LIN {X 0,Y 325.201,Z 458.699,A -85,B 0,C 180,E1 -14842.55,E2 -14842.55} C_VEL
LIN {X 0,Y 325.198,Z 460.508,A -85,B 0,C 180,E1 -14843.797,E2 -14843.797} C_VEL
LIN {X 0,Y 325.238,Z 461.898,A -85,B 0,C 180,E1 -14845.041,E2 -14845.041} C_VEL
LIN {X 0,Y 325.475,Z 463.331,A -85,B 0,C 180,E1 -14847.525,E2 -14847.525} C_VEL
LIN {X 0,Y 325.603,Z 463.425,A -85,B 0,C 180,E1 -14848.763,E2 -14848.763} C_VEL
LIN {X 0,Y 325.577,Z 463.02,A -85,B 0,C 180,E1 -14850,E2 -14850} C_VEL
LIN {X 0,Y 325.621,Z 461.713,A -85,B 0,C 180,E1 -14852.474,E2 -14852.474} C_VEL
LIN {X 0,Y 325.409,Z 460.927,A -85,B 0,C 180,E1 -14853.715,E2 -14853.715} C_VEL
LIN {X 0,Y 325.339,Z 458.485,A -85,B 0,C 180,E1 -14855.579,E2 -14855.579} C_VEL
LIN {X 0,Y 325.419,Z 455.521,A -85,B 0,C 180,E1 -14856.994,E2 -14856.994} C_VEL
LIN {X 0,Y 325.54,Z 450.546,A -85,B 0,C 180,E1 -14858.692,E2 -14858.692} C_VEL
LIN {X 0,Y 325.777,Z 444.462,A -85,B 0,C 180,E1 -14860.252,E2 -14860.252} C_VEL
LIN {X 0,Y 326.095,Z 438.305,A -85,B 0,C 180,E1 -14861.499,E2 -14861.499} C_VEL
LIN {X 0,Y 326.625,Z 429.473,A -85,B 0,C 180,E1 -14862.899,E2 -14862.899} C_VEL
LIN {X 0,Y 326.943,Z 420.656,A -85,B 0,C 180,E1 -14863.995,E2 -14863.995} C_VEL
LIN {X 0,Y 327.306,Z 414.872,A -85,B 0,C 180,E1 -14864.614,E2 -14864.614} C_VEL
LIN {X 0,Y 327.995,Z 404.103,A -85,B 0,C 180,E1 -14865.823,E2 -14865.823} C_VEL
LIN {X 0,Y 328.456,Z 394.191,A -85,B 0,C 180,E1 -14866.71,E2 -14866.71} C_VEL
LIN {X 0,Y 327.545,Z 382.063,A -85,B 0,C 180,E1 -14867.562,E2 -14867.562} C_VEL
LIN {X 0,Y 327.132,Z 375.822,A -85,B 0,C 180,E1 -14867.908,E2 -14867.908} C_VEL
LIN {X 0,Y 327.626,Z 366.768,A -85,B 0,C 180,E1 -14869.042,E2 -14869.042} C_VEL
LIN {X 0,Y 327.17,Z 358.001,A -85,B 0,C 180,E1 -14870.43,E2 -14870.43} C_VEL
LIN {X 0,Y 328.784,Z 345.205,A -85,B 0,C 180,E1 -14874.635,E2 -14874.635} C_VEL
LIN {X 0,Y 330.645,Z 333.295,A -85,B 0,C 180,E1 -14878.571,E2 -14878.571} C_VEL
LIN {X 0,Y 331.363,Z 329.074,A -85,B 0,C 180,E1 -14879.977,E2 -14879.977} C_VEL
LIN {X 0,Y 331.435,Z 327.269,A -85,B 0,C 180,E1 -14880.592,E2 -14880.592} C_VEL
LIN {X 0,Y 329.253,Z 316.724,A -85,B 0,C 180,E1 -14884.447,E2 -14884.447} C_VEL
LIN {X 0,Y 326.968,Z 305.312,A -85,B 0,C 180,E1 -14888.825,E2 -14888.825} C_VEL
LIN {X 0,Y 326.92,Z 305.233,A -85,B 0,C 180,E1 -14891.792,E2 -14891.792} C_VEL
LIN {X 0,Y 327.446,Z 306.47,A -85,B 0,C 180,E1 -14895.096,E2 -14895.096} C_VEL
LIN {X 0,Y 328.262,Z 309.046,A -85,B 0,C 180,E1 -14898.534,E2 -14898.534} C_VEL
LIN {X 0,Y 329.377,Z 312.876,A -85,B 0,C 180,E1 -14902.137,E2 -14902.137} C_VEL
LIN {X 0,Y 330.222,Z 316.406,A -85,B 0,C 180,E1 -14904.925,E2 -14904.925} C_VEL
LIN {X 0,Y 330.999,Z 321.163,A -85,B 0,C 180,E1 -14908.137,E2 -14908.137} C_VEL
LIN {X 0,Y 331.171,Z 324.386,A -85,B 0,C 180,E1 -14910.085,E2 -14910.085} C_VEL
LIN {X 0,Y 330.472,Z 330.636,A -85,B 0,C 180,E1 -14913.473,E2 -14913.473} C_VEL
LIN {X 0,Y 329.774,Z 338.112,A -85,B 0,C 180,E1 -14917.441,E2 -14917.441} C_VEL
LIN {X 0,Y 329.205,Z 345.556,A -85,B 0,C 180,E1 -14921.322,E2 -14921.322} C_VEL
LIN {X 0,Y 328.9,Z 351.017,A -85,B 0,C 180,E1 -14924.127,E2 -14924.127} C_VEL
LIN {X 0,Y 332.084,Z 361.27,A -85,B 0,C 180,E1 -14925.287,E2 -14925.287} C_VEL
LIN {X 0,Y 333.261,Z 367.816,A -85,B 0,C 180,E1 -14926.104,E2 -14926.104} C_VEL
LIN {X 0,Y 332.238,Z 376.783,A -85,B 0,C 180,E1 -14927.226,E2 -14927.226} C_VEL
LIN {X 0,Y 331.076,Z 383.941,A -85,B 0,C 180,E1 -14928.364,E2 -14928.364} C_VEL
LIN {X 0,Y 330.119,Z 389.732,A -85,B 0,C 180,E1 -14929.573,E2 -14929.573} C_VEL
LIN {X 0,Y 329.305,Z 394.315,A -85,B 0,C 180,E1 -14930.788,E2 -14930.788} C_VEL
LIN {X 0,Y 328.522,Z 397.947,A -85,B 0,C 180,E1 -14932.005,E2 -14932.005} C_VEL
LIN {X 0,Y 327.856,Z 400.687,A -85,B 0,C 180,E1 -14933.228,E2 -14933.228} C_VEL
LIN {X 0,Y 326.757,Z 403.34,A -85,B 0,C 180,E1 -14935.063,E2 -14935.063} C_VEL
LIN {X 0,Y 326.193,Z 404.249,A -85,B 0,C 180,E1 -14936.292,E2 -14936.292} C_VEL
LIN {X 0,Y 325.862,Z 404.462,A -85,B 0,C 180,E1 -14937.526,E2 -14937.526} C_VEL
LIN {X 0,Y 325.68,Z 403.978,A -85,B 0,C 180,E1 -14938.762,E2 -14938.762} C_VEL
LIN {X 0,Y 325.531,Z 402.803,A -85,B 0,C 180,E1 -14939.998,E2 -14939.998} C_VEL
LIN {X 0,Y 325.509,Z 399.647,A -85,B 0,C 180,E1 -14941.854,E2 -14941.854} C_VEL
LIN {X 0,Y 325.609,Z 396.615,A -85,B 0,C 180,E1 -14943.092,E2 -14943.092} C_VEL
LIN {X 0,Y 325.781,Z 391.513,A -85,B 0,C 180,E1 -14944.639,E2 -14944.639} C_VEL
LIN {X 0,Y 326.058,Z 386.269,A -85,B 0,C 180,E1 -14945.875,E2 -14945.875} C_VEL
LIN {X 0,Y 326.233,Z 378.87,A -85,B 0,C 180,E1 -14947.237,E2 -14947.237} C_VEL
LIN {X 0,Y 326.433,Z 371.108,A -85,B 0,C 180,E1 -14948.354,E2 -14948.354} C_VEL
LIN {X 0,Y 326.671,Z 362.647,A -85,B 0,C 180,E1 -14949.284,E2 -14949.284} C_VEL
LIN {X 0,Y 326.921,Z 353.507,A -85,B 0,C 180,E1 -14950.058,E2 -14950.058} C_VEL
LIN {X 0,Y 326.042,Z 345.613,A -85,B 0,C 180,E1 -14950.556,E2 -14950.556} C_VEL
LIN {X 0,Y 326.165,Z 337.653,A -85,B 0,C 180,E1 -14954.155,E2 -14954.155} C_VEL
LIN {X 0,Y 326.232,Z 328.045,A -85,B 0,C 180,E1 -14958.578,E2 -14958.578} C_VEL
LIN {X 0,Y 326.347,Z 320.299,A -85,B 0,C 180,E1 -14962.176,E2 -14962.176} C_VEL
LIN {X 0,Y 326.533,Z 313.209,A -85,B 0,C 180,E1 -14965.495,E2 -14965.495} C_VEL
LIN {X 0,Y 326.706,Z 305.841,A -85,B 0,C 180,E1 -14968.946,E2 -14968.946} C_VEL
LIN {X 0,Y 326.794,Z 303.776,A -85,B 0,C 180,E1 -14969.961,E2 -14969.961} C_VEL
LIN {X 0,Y 326.602,Z 303.799,A -85,B 0,C 180,E1 -14974.018,E2 -14974.018} C_VEL
LIN {X 0,Y 326.617,Z 303.802,A -85,B 0,C 180,E1 -14977.236,E2 -14977.236} C_VEL
LIN {X 0,Y 326.538,Z 303.812,A -85,B 0,C 180,E1 -14981.123,E2 -14981.123} C_VEL
LIN {X 0,Y 326.554,Z 303.807,A -85,B 0,C 180,E1 -14983.524,E2 -14983.524} C_VEL
LIN {X 0,Y 326.568,Z 303.808,A -85,B 0,C 180,E1 -14987.027,E2 -14987.027} C_VEL
LIN {X 0,Y 326.604,Z 303.804,A -85,B 0,C 180,E1 -14990.771,E2 -14990.771} C_VEL
LIN {X 0,Y 326.605,Z 303.802,A -85,B 0,C 180,E1 -14994.479,E2 -14994.479} C_VEL
LIN {X 0,Y 326.599,Z 303.8,A -85,B 0,C 180,E1 -14997.454,E2 -14997.454} C_VEL
LIN {X 0,Y 326.651,Z 303.796,A -85,B 0,C 180,E1 -15000.34,E2 -15000.34} C_VEL
LIN {X 0,Y 326.68,Z 303.795,A -85,B 0,C 180,E1 -15004.515,E2 -15004.515} C_VEL
LIN {X 0,Y 326.636,Z 303.8,A -85,B 0,C 180,E1 -15008.544,E2 -15008.544} C_VEL
LIN {X 0,Y 326.733,Z 303.783,A -85,B 0,C 180,E1 -15011.177,E2 -15011.177} C_VEL
LIN {X 0,Y 326.752,Z 303.78,A -85,B 0,C 180,E1 -15015.433,E2 -15015.433} C_VEL
LIN {X 0,Y 326.746,Z 303.782,A -85,B 0,C 180,E1 -15018.838,E2 -15018.838} C_VEL
LIN {X 0,Y 326.902,Z 303.764,A -85,B 0,C 180,E1 -15022.589,E2 -15022.589} C_VEL
LIN {X 0,Y 326.74,Z 303.782,A -85,B 0,C 180,E1 -15025.064,E2 -15025.064} C_VEL
LIN {X 0,Y 326.998,Z 303.751,A -85,B 0,C 180,E1 -15027.536,E2 -15027.536} C_VEL
LIN {X 0,Y 327.016,Z 303.748,A -85,B 0,C 180,E1 -15031.231,E2 -15031.231} C_VEL
LIN {X 0,Y 326.745,Z 303.785,A -85,B 0,C 180,E1 -15033.7,E2 -15033.7} C_VEL
LIN {X 0,Y 326.932,Z 303.761,A -85,B 0,C 180,E1 -15036.17,E2 -15036.17} C_VEL
LIN {X 0,Y 326.771,Z 303.782,A -85,B 0,C 180,E1 -15039.908,E2 -15039.908} C_VEL
LIN {X 0,Y 326.747,Z 303.787,A -85,B 0,C 180,E1 -15043.686,E2 -15043.686} C_VEL
LIN {X 0,Y 326.689,Z 303.793,A -85,B 0,C 180,E1 -15047.529,E2 -15047.529} C_VEL
LIN {X 0,Y 326.657,Z 303.793,A -85,B 0,C 180,E1 -15050.135,E2 -15050.135} C_VEL
LIN {X 0,Y 326.642,Z 303.795,A -85,B 0,C 180,E1 -15054.13,E2 -15054.13} C_VEL
LIN {X 0,Y 326.675,Z 303.791,A -85,B 0,C 180,E1 -15056.859,E2 -15056.859} C_VEL
LIN {X 0,Y 326.629,Z 303.796,A -85,B 0,C 180,E1 -15060.612,E2 -15060.612} C_VEL
LIN {X 0,Y 326.598,Z 303.8,A -85,B 0,C 180,E1 -15064.021,E2 -15064.021} C_VEL
LIN {X 0,Y 326.621,Z 303.802,A -85,B 0,C 180,E1 -15067.24,E2 -15067.24} C_VEL
LIN {X 0,Y 326.57,Z 303.808,A -85,B 0,C 180,E1 -15071.133,E2 -15071.133} C_VEL
LIN {X 0,Y 326.52,Z 303.813,A -85,B 0,C 180,E1 -15074.744,E2 -15074.744} C_VEL
LIN {X 0,Y 326.555,Z 303.805,A -85,B 0,C 180,E1 -15078.154,E2 -15078.154} C_VEL
LIN {X 0,Y 326.575,Z 303.804,A -85,B 0,C 180,E1 -15081.387,E2 -15081.387} C_VEL
LIN {X 0,Y 326.614,Z 303.803,A -85,B 0,C 180,E1 -15084.853,E2 -15084.853} C_VEL
LIN {X 0,Y 326.811,Z 303.868,A -85,B 0,C 180,E1 -15088.48,E2 -15088.48} C_VEL
LIN {X 0,Y 326.946,Z 306.82,A -85,B 0,C 180,E1 -15090.372,E2 -15090.372} C_VEL
LIN {X 0,Y 326.556,Z 312.39,A -85,B 0,C 180,E1 -15093.822,E2 -15093.822} C_VEL
LIN {X 0,Y 326.169,Z 319.095,A -85,B 0,C 180,E1 -15097.9,E2 -15097.9} C_VEL
LIN {X 0,Y 325.915,Z 324.514,A -85,B 0,C 180,E1 -15101.13,E2 -15101.13} C_VEL
LIN {X 0,Y 325.724,Z 328.884,A -85,B 0,C 180,E1 -15103.692,E2 -15103.692} C_VEL
LIN {X 0,Y 325.001,Z 330.075,A -85,B 0,C 180,E1 -15104.347,E2 -15104.347} C_VEL
LIN {X 0,Y 322.085,Z 332.054,A -85,B 0,C 180,E1 -15105.362,E2 -15105.362} C_VEL
LIN {X 0,Y 319.171,Z 334.053,A -85,B 0,C 180,E1 -15106.394,E2 -15106.394} C_VEL
LIN {X 0,Y 318.479,Z 335.258,A -85,B 0,C 180,E1 -15107.067,E2 -15107.067} C_VEL
LIN {X 0,Y 318.465,Z 336.636,A -85,B 0,C 180,E1 -15107.86,E2 -15107.86} C_VEL
LIN {X 0,Y 319.617,Z 348.07,A -85,B 0,C 180,E1 -15108.668,E2 -15108.668} C_VEL
LIN {X 0,Y 320.397,Z 354.645,A -85,B 0,C 180,E1 -15109.256,E2 -15109.256} C_VEL
LIN {X 0,Y 319.903,Z 364.882,A -85,B 0,C 180,E1 -15110.358,E2 -15110.358} C_VEL
LIN {X 0,Y 319.519,Z 374.615,A -85,B 0,C 180,E1 -15111.706,E2 -15111.706} C_VEL
LIN {X 0,Y 319.21,Z 382.258,A -85,B 0,C 180,E1 -15113.047,E2 -15113.047} C_VEL
LIN {X 0,Y 318.893,Z 389.43,A -85,B 0,C 180,E1 -15114.627,E2 -15114.627} C_VEL
LIN {X 0,Y 318.581,Z 395.045,A -85,B 0,C 180,E1 -15116.207,E2 -15116.207} C_VEL
LIN {X 0,Y 318.433,Z 400.056,A -85,B 0,C 180,E1 -15118.104,E2 -15118.104} C_VEL
LIN {X 0,Y 318.484,Z 403.441,A -85,B 0,C 180,E1 -15120.002,E2 -15120.002} C_VEL
LIN {X 0,Y 318.636,Z 404.864,A -85,B 0,C 180,E1 -15121.265,E2 -15121.265} C_VEL
LIN {X 0,Y 318.85,Z 405.644,A -85,B 0,C 180,E1 -15122.528,E2 -15122.528} C_VEL
LIN {X 0,Y 319.196,Z 405.78,A -85,B 0,C 180,E1 -15123.789,E2 -15123.789} C_VEL
LIN {X 0,Y 319.771,Z 405.275,A -85,B 0,C 180,E1 -15125.045,E2 -15125.045} C_VEL
LIN {X 0,Y 320.449,Z 404.147,A -85,B 0,C 180,E1 -15126.297,E2 -15126.297} C_VEL
LIN {X 0,Y 321.74,Z 401.238,A -85,B 0,C 180,E1 -15128.164,E2 -15128.164} C_VEL
LIN {X 0,Y 323.183,Z 396.853,A -85,B 0,C 180,E1 -15130.02,E2 -15130.02} C_VEL
LIN {X 0,Y 324.589,Z 391.903,A -85,B 0,C 180,E1 -15131.555,E2 -15131.555} C_VEL
LIN {X 0,Y 326.271,Z 385.501,A -85,B 0,C 180,E1 -15133.073,E2 -15133.073} C_VEL
LIN {X 0,Y 328.143,Z 377.5,A -85,B 0,C 180,E1 -15134.577,E2 -15134.577} C_VEL
LIN {X 0,Y 329.055,Z 372.691,A -85,B 0,C 180,E1 -15135.338,E2 -15135.338} C_VEL
LIN {X 0,Y 328.549,Z 366.669,A -85,B 0,C 180,E1 -15136.371,E2 -15136.371} C_VEL
LIN {X 0,Y 326.537,Z 357.316,A -85,B 0,C 180,E1 -15137.935,E2 -15137.935} C_VEL
LIN {X 0,Y 323.137,Z 347.004,A -85,B 0,C 180,E1 -15139.608,E2 -15139.608} C_VEL
LIN {X 0,Y 321.875,Z 343.462,A -85,B 0,C 180,E1 -15140.22,E2 -15140.22} C_VEL
LIN {X 0,Y 322.799,Z 339.37,A -85,B 0,C 180,E1 -15143.875,E2 -15143.875} C_VEL
LIN {X 0,Y 323.719,Z 336.122,A -85,B 0,C 180,E1 -15147.125,E2 -15147.125} C_VEL
LIN {X 0,Y 324.569,Z 333.676,A -85,B 0,C 180,E1 -15149.987,E2 -15149.987} C_VEL
LIN {X 0,Y 325.098,Z 331.86,A -85,B 0,C 180,E1 -15152.716,E2 -15152.716} C_VEL
LIN {X 0,Y 325.329,Z 330.489,A -85,B 0,C 180,E1 -15155.683,E2 -15155.683} C_VEL
LIN {X 0,Y 325.489,Z 329.814,A -85,B 0,C 180,E1 -15158.984,E2 -15158.984} C_VEL
LIN {X 0,Y 325.709,Z 329.954,A -85,B 0,C 180,E1 -15161.984,E2 -15161.984} C_VEL
LIN {X 0,Y 326.092,Z 331.016,A -85,B 0,C 180,E1 -15165.336,E2 -15165.336} C_VEL
LIN {X 0,Y 326.701,Z 333.227,A -85,B 0,C 180,E1 -15168.846,E2 -15168.846} C_VEL
LIN {X 0,Y 327.276,Z 335.665,A -85,B 0,C 180,E1 -15171.482,E2 -15171.482} C_VEL
LIN {X 0,Y 328.152,Z 339.585,A -85,B 0,C 180,E1 -15174.672,E2 -15174.672} C_VEL
LIN {X 0,Y 328.855,Z 343.249,A -85,B 0,C 180,E1 -15177.115,E2 -15177.115} C_VEL
LIN {X 0,Y 328.826,Z 345.636,A -85,B 0,C 180,E1 -15178.412,E2 -15178.412} C_VEL
LIN {X 0,Y 326.738,Z 351.583,A -85,B 0,C 180,E1 -15181.055,E2 -15181.055} C_VEL
LIN {X 0,Y 324.056,Z 361.03,A -85,B 0,C 180,E1 -15184.831,E2 -15184.831} C_VEL
LIN {X 0,Y 326.737,Z 372.97,A -85,B 0,C 180,E1 -15185.96,E2 -15185.96} C_VEL
LIN {X 0,Y 328.385,Z 385.404,A -85,B 0,C 180,E1 -15187.189,E2 -15187.189} C_VEL
LIN {X 0,Y 328.621,Z 394.021,A -85,B 0,C 180,E1 -15188.084,E2 -15188.084} C_VEL
LIN {X 0,Y 327.755,Z 404.734,A -85,B 0,C 180,E1 -15189.28,E2 -15189.28} C_VEL
LIN {X 0,Y 325.502,Z 416.387,A -85,B 0,C 180,E1 -15190.776,E2 -15190.776} C_VEL
LIN {X 0,Y 323.559,Z 425.786,A -85,B 0,C 180,E1 -15192.296,E2 -15192.296} C_VEL
LIN {X 0,Y 321.827,Z 434.424,A -85,B 0,C 180,E1 -15194.013,E2 -15194.013} C_VEL
LIN {X 0,Y 320.493,Z 441.391,A -85,B 0,C 180,E1 -15195.718,E2 -15195.718} C_VEL
LIN {X 0,Y 319.161,Z 448.602,A -85,B 0,C 180,E1 -15197.925,E2 -15197.925} C_VEL
LIN {X 0,Y 318.477,Z 453.47,A -85,B 0,C 180,E1 -15199.832,E2 -15199.832} C_VEL
LIN {X 0,Y 318.176,Z 457.251,A -85,B 0,C 180,E1 -15201.745,E2 -15201.745} C_VEL
LIN {X 0,Y 318.114,Z 460.19,A -85,B 0,C 180,E1 -15203.82,E2 -15203.82} C_VEL
LIN {X 0,Y 318.207,Z 462.144,A -85,B 0,C 180,E1 -15206.201,E2 -15206.201} C_VEL
LIN {X 0,Y 318.406,Z 462.61,A -85,B 0,C 180,E1 -15207.47,E2 -15207.47} C_VEL
LIN {X 0,Y 318.557,Z 462.602,A -85,B 0,C 180,E1 -15208.736,E2 -15208.736} C_VEL
LIN {X 0,Y 318.535,Z 462.136,A -85,B 0,C 180,E1 -15210,E2 -15210} C_VEL
LIN {X 0,Y 318.581,Z 461.254,A -85,B 0,C 180,E1 -15211.264,E2 -15211.264} C_VEL
LIN {X 0,Y 318.542,Z 461.03,A -85,B 0,C 180,E1 -15212.529,E2 -15212.529} C_VEL
LIN {X 0,Y 318.315,Z 460.375,A -85,B 0,C 180,E1 -15213.798,E2 -15213.798} C_VEL
LIN {X 0,Y 318.248,Z 458.067,A -85,B 0,C 180,E1 -15215.703,E2 -15215.703} C_VEL
LIN {X 0,Y 318.334,Z 455.796,A -85,B 0,C 180,E1 -15216.911,E2 -15216.911} C_VEL
LIN {X 0,Y 318.43,Z 452.507,A -85,B 0,C 180,E1 -15218.248,E2 -15218.248} C_VEL
LIN {X 0,Y 318.659,Z 447.294,A -85,B 0,C 180,E1 -15219.842,E2 -15219.842} C_VEL
LIN {X 0,Y 319.046,Z 440.563,A -85,B 0,C 180,E1 -15221.435,E2 -15221.435} C_VEL
LIN {X 0,Y 319.58,Z 433.596,A -85,B 0,C 180,E1 -15222.704,E2 -15222.704} C_VEL
LIN {X 0,Y 320.171,Z 424.987,A -85,B 0,C 180,E1 -15223.973,E2 -15223.973} C_VEL
LIN {X 0,Y 320.603,Z 416.959,A -85,B 0,C 180,E1 -15224.889,E2 -15224.889} C_VEL
LIN {X 0,Y 320.859,Z 408.42,A -85,B 0,C 180,E1 -15225.678,E2 -15225.678} C_VEL
LIN {X 0,Y 321.282,Z 399.098,A -85,B 0,C 180,E1 -15226.342,E2 -15226.342} C_VEL
LIN {X 0,Y 321.27,Z 392.257,A -85,B 0,C 180,E1 -15226.931,E2 -15226.931} C_VEL
LIN {X 0,Y 320.643,Z 384.318,A -85,B 0,C 180,E1 -15227.541,E2 -15227.541} C_VEL
LIN {X 0,Y 321.076,Z 373.539,A -85,B 0,C 180,E1 -15228.9,E2 -15228.9} C_VEL
LIN {X 0,Y 321.416,Z 367.768,A -85,B 0,C 180,E1 -15229.677,E2 -15229.677} C_VEL
LIN {X 0,Y 320.631,Z 356.741,A -85,B 0,C 180,E1 -15231.54,E2 -15231.54} C_VEL
LIN {X 0,Y 320.711,Z 353.082,A -85,B 0,C 180,E1 -15232.206,E2 -15232.206} C_VEL
LIN {X 0,Y 322.675,Z 339.681,A -85,B 0,C 180,E1 -15236.745,E2 -15236.745} C_VEL
LIN {X 0,Y 324.372,Z 329.417,A -85,B 0,C 180,E1 -15240.248,E2 -15240.248} C_VEL
LIN {X 0,Y 324.01,Z 326.296,A -85,B 0,C 180,E1 -15241.371,E2 -15241.371} C_VEL
LIN {X 0,Y 321.838,Z 315.95,A -85,B 0,C 180,E1 -15245.272,E2 -15245.272} C_VEL
LIN {X 0,Y 320.813,Z 310.811,A -85,B 0,C 180,E1 -15247.34,E2 -15247.34} C_VEL
LIN {X 0,Y 321.336,Z 309.451,A -85,B 0,C 180,E1 -15249.366,E2 -15249.366} C_VEL
LIN {X 0,Y 321.211,Z 309.612,A -85,B 0,C 180,E1 -15252.709,E2 -15252.709} C_VEL
LIN {X 0,Y 321.607,Z 310.739,A -85,B 0,C 180,E1 -15255.628,E2 -15255.628} C_VEL
LIN {X 0,Y 322.32,Z 313.311,A -85,B 0,C 180,E1 -15259.145,E2 -15259.145} C_VEL
LIN {X 0,Y 323.261,Z 316.722,A -85,B 0,C 180,E1 -15262.5,E2 -15262.5} C_VEL
LIN {X 0,Y 323.697,Z 318.563,A -85,B 0,C 180,E1 -15264.11,E2 -15264.11} C_VEL
LIN {X 0,Y 324.428,Z 323.404,A -85,B 0,C 180,E1 -15267.656,E2 -15267.656} C_VEL
LIN {X 0,Y 324.61,Z 327.062,A -85,B 0,C 180,E1 -15270,E2 -15270} C_VEL
LIN {X 0,Y 323.814,Z 333.536,A -85,B 0,C 180,E1 -15273.58,E2 -15273.58} C_VEL
LIN {X 0,Y 323.017,Z 340.963,A -85,B 0,C 180,E1 -15277.618,E2 -15277.618} C_VEL
LIN {X 0,Y 322.427,Z 348.394,A -85,B 0,C 180,E1 -15281.574,E2 -15281.574} C_VEL
LIN {X 0,Y 322.192,Z 351.989,A -85,B 0,C 180,E1 -15283.439,E2 -15283.439} C_VEL
LIN {X 0,Y 324.917,Z 360.301,A -85,B 0,C 180,E1 -15284.423,E2 -15284.423} C_VEL
LIN {X 0,Y 326.726,Z 368.156,A -85,B 0,C 180,E1 -15285.46,E2 -15285.46} C_VEL
LIN {X 0,Y 326.709,Z 371.356,A -85,B 0,C 180,E1 -15285.852,E2 -15285.852} C_VEL
LIN {X 0,Y 325.558,Z 379.854,A -85,B 0,C 180,E1 -15287.023,E2 -15287.023} C_VEL
LIN {X 0,Y 324.376,Z 386.132,A -85,B 0,C 180,E1 -15288.12,E2 -15288.12} C_VEL
LIN {X 0,Y 323.166,Z 392.806,A -85,B 0,C 180,E1 -15289.663,E2 -15289.663} C_VEL
LIN {X 0,Y 322.023,Z 397.743,A -85,B 0,C 180,E1 -15291.211,E2 -15291.211} C_VEL
LIN {X 0,Y 321.174,Z 400.745,A -85,B 0,C 180,E1 -15292.454,E2 -15292.454} C_VEL
LIN {X 0,Y 320.443,Z 402.945,A -85,B 0,C 180,E1 -15293.703,E2 -15293.703} C_VEL
LIN {X 0,Y 319.763,Z 404.411,A -85,B 0,C 180,E1 -15294.955,E2 -15294.955} C_VEL
LIN {X 0,Y 319.169,Z 405.168,A -85,B 0,C 180,E1 -15296.211,E2 -15296.211} C_VEL
LIN {X 0,Y 318.827,Z 405.216,A -85,B 0,C 180,E1 -15297.472,E2 -15297.472} C_VEL
LIN {X 0,Y 318.62,Z 404.576,A -85,B 0,C 180,E1 -15298.734,E2 -15298.734} C_VEL
LIN {X 0,Y 318.411,Z 402.308,A -85,B 0,C 180,E1 -15300.631,E2 -15300.631} C_VEL
LIN {X 0,Y 318.44,Z 399.914,A -85,B 0,C 180,E1 -15301.895,E2 -15301.895} C_VEL
LIN {X 0,Y 318.53,Z 396.7,A -85,B 0,C 180,E1 -15303.16,E2 -15303.16} C_VEL
LIN {X 0,Y 318.71,Z 391.336,A -85,B 0,C 180,E1 -15304.742,E2 -15304.742} C_VEL
LIN {X 0,Y 319.001,Z 385.885,A -85,B 0,C 180,E1 -15306.005,E2 -15306.005} C_VEL
LIN {X 0,Y 319.158,Z 377.987,A -85,B 0,C 180,E1 -15307.416,E2 -15307.416} C_VEL
LIN {X 0,Y 319.392,Z 369.888,A -85,B 0,C 180,E1 -15308.54,E2 -15308.54} C_VEL
LIN {X 0,Y 319.593,Z 361.028,A -85,B 0,C 180,E1 -15309.491,E2 -15309.491} C_VEL
LIN {X 0,Y 319.784,Z 353.253,A -85,B 0,C 180,E1 -15310.125,E2 -15310.125} C_VEL
LIN {X 0,Y 318.982,Z 346.194,A -85,B 0,C 180,E1 -15310.591,E2 -15310.591} C_VEL
LIN {X 0,Y 319.101,Z 338.081,A -85,B 0,C 180,E1 -15314.286,E2 -15314.286} C_VEL
LIN {X 0,Y 319.154,Z 330.149,A -85,B 0,C 180,E1 -15317.954,E2 -15317.954} C_VEL
LIN {X 0,Y 319.297,Z 323.005,A -85,B 0,C 180,E1 -15321.294,E2 -15321.294} C_VEL
LIN {X 0,Y 319.509,Z 313.886,A -85,B 0,C 180,E1 -15325.598,E2 -15325.598} C_VEL
LIN {X 0,Y 319.759,Z 304.652,A -85,B 0,C 180,E1 -15329.999,E2 -15329.999} C_VEL
LIN {X 0,Y 319.571,Z 304.679,A -85,B 0,C 180,E1 -15333.351,E2 -15333.351} C_VEL
LIN {X 0,Y 319.55,Z 304.678,A -85,B 0,C 180,E1 -15336.426,E2 -15336.426} C_VEL
LIN {X 0,Y 319.521,Z 304.682,A -85,B 0,C 180,E1 -15339.66,E2 -15339.66} C_VEL
LIN {X 0,Y 319.513,Z 304.684,A -85,B 0,C 180,E1 -15343.459,E2 -15343.459} C_VEL
LIN {X 0,Y 319.546,Z 304.683,A -85,B 0,C 180,E1 -15347.015,E2 -15347.015} C_VEL
LIN {X 0,Y 319.539,Z 304.68,A -85,B 0,C 180,E1 -15350.37,E2 -15350.37} C_VEL
LIN {X 0,Y 319.551,Z 304.678,A -85,B 0,C 180,E1 -15353.571,E2 -15353.571} C_VEL
LIN {X 0,Y 319.568,Z 304.68,A -85,B 0,C 180,E1 -15356.685,E2 -15356.685} C_VEL
LIN {X 0,Y 319.582,Z 304.673,A -85,B 0,C 180,E1 -15359.615,E2 -15359.615} C_VEL
LIN {X 0,Y 319.6,Z 304.676,A -85,B 0,C 180,E1 -15362.497,E2 -15362.497} C_VEL
LIN {X 0,Y 319.594,Z 304.672,A -85,B 0,C 180,E1 -15365.303,E2 -15365.303} C_VEL
LIN {X 0,Y 319.586,Z 304.675,A -85,B 0,C 180,E1 -15368.047,E2 -15368.047} C_VEL
LIN {X 0,Y 319.678,Z 304.663,A -85,B 0,C 180,E1 -15370.961,E2 -15370.961} C_VEL
LIN {X 0,Y 319.72,Z 304.656,A -85,B 0,C 180,E1 -15375.275,E2 -15375.275} C_VEL
LIN {X 0,Y 319.703,Z 304.661,A -85,B 0,C 180,E1 -15378.589,E2 -15378.589} C_VEL
LIN {X 0,Y 319.841,Z 304.644,A -85,B 0,C 180,E1 -15382.424,E2 -15382.424} C_VEL
LIN {X 0,Y 319.709,Z 304.658,A -85,B 0,C 180,E1 -15384.955,E2 -15384.955} C_VEL
LIN {X 0,Y 319.945,Z 304.629,A -85,B 0,C 180,E1 -15387.482,E2 -15387.482} C_VEL
LIN {X 0,Y 319.985,Z 304.624,A -85,B 0,C 180,E1 -15391.259,E2 -15391.259} C_VEL
LIN {X 0,Y 319.695,Z 304.664,A -85,B 0,C 180,E1 -15393.781,E2 -15393.781} C_VEL
LIN {X 0,Y 319.889,Z 304.637,A -85,B 0,C 180,E1 -15396.307,E2 -15396.307} C_VEL
LIN {X 0,Y 319.723,Z 304.658,A -85,B 0,C 180,E1 -15400.128,E2 -15400.128} C_VEL
LIN {X 0,Y 319.721,Z 304.659,A -85,B 0,C 180,E1 -15403.993,E2 -15403.993} C_VEL
LIN {X 0,Y 319.648,Z 304.668,A -85,B 0,C 180,E1 -15407.928,E2 -15407.928} C_VEL
LIN {X 0,Y 319.607,Z 304.67,A -85,B 0,C 180,E1 -15410.6,E2 -15410.6} C_VEL
LIN {X 0,Y 319.56,Z 304.68,A -85,B 0,C 180,E1 -15413.32,E2 -15413.32} C_VEL
LIN {X 0,Y 319.625,Z 304.669,A -85,B 0,C 180,E1 -15416.089,E2 -15416.089} C_VEL
LIN {X 0,Y 319.58,Z 304.676,A -85,B 0,C 180,E1 -15418.935,E2 -15418.935} C_VEL
LIN {X 0,Y 319.523,Z 304.682,A -85,B 0,C 180,E1 -15421.863,E2 -15421.863} C_VEL
LIN {X 0,Y 319.572,Z 304.677,A -85,B 0,C 180,E1 -15425.545,E2 -15425.545} C_VEL
LIN {X 0,Y 319.55,Z 304.677,A -85,B 0,C 180,E1 -15428.011,E2 -15428.011} C_VEL
LIN {X 0,Y 319.518,Z 304.683,A -85,B 0,C 180,E1 -15431.599,E2 -15431.599} C_VEL
LIN {X 0,Y 319.48,Z 304.689,A -85,B 0,C 180,E1 -15435.259,E2 -15435.259} C_VEL
LIN {X 0,Y 319.498,Z 304.685,A -85,B 0,C 180,E1 -15438.409,E2 -15438.409} C_VEL
LIN {X 0,Y 319.525,Z 304.681,A -85,B 0,C 180,E1 -15441.988,E2 -15441.988} C_VEL
LIN {X 0,Y 319.558,Z 304.679,A -85,B 0,C 180,E1 -15445.126,E2 -15445.126} C_VEL
LIN {X 0,Y 319.768,Z 304.717,A -85,B 0,C 180,E1 -15448.411,E2 -15448.411} C_VEL
LIN {X 0,Y 319.896,Z 307.77,A -85,B 0,C 180,E1 -15450.377,E2 -15450.377} C_VEL
LIN {X 0,Y 319.484,Z 313.355,A -85,B 0,C 180,E1 -15453.901,E2 -15453.901} C_VEL
LIN {X 0,Y 319.09,Z 320.032,A -85,B 0,C 180,E1 -15458.013,E2 -15458.013} C_VEL
LIN {X 0,Y 318.822,Z 325.676,A -85,B 0,C 180,E1 -15461.42,E2 -15461.42} C_VEL
LIN {X 0,Y 318.554,Z 332.238,A -85,B 0,C 180,E1 -15465.304,E2 -15465.304} C_VEL
LIN {X 0,Y 318.479,Z 335.258,A -85,B 0,C 180,E1 -15467.067,E2 -15467.067} C_VEL
LIN {X 0,Y 318.357,Z 337.059,A -85,B 0,C 180,E1 -15467.587,E2 -15467.587} C_VEL
LIN {X 0,Y 318.052,Z 339.817,A -85,B 0,C 180,E1 -15467.975,E2 -15467.975} C_VEL
LIN {X 0,Y 317.421,Z 343.988,A -85,B 0,C 180,E1 -15468.319,E2 -15468.319} C_VEL
LIN {X 0,Y 316.006,Z 350.409,A -85,B 0,C 180,E1 -15468.801,E2 -15468.801} C_VEL
LIN {X 0,Y 313.416,Z 359.289,A -85,B 0,C 180,E1 -15469.622,E2 -15469.622} C_VEL
LIN {X 0,Y 312.97,Z 362.174,A -85,B 0,C 180,E1 -15469.95,E2 -15469.95} C_VEL
LIN {X 0,Y 312.534,Z 372.219,A -85,B 0,C 180,E1 -15471.272,E2 -15471.272} C_VEL
LIN {X 0,Y 312.167,Z 380.05,A -85,B 0,C 180,E1 -15472.565,E2 -15472.565} C_VEL
LIN {X 0,Y 311.925,Z 387.861,A -85,B 0,C 180,E1 -15474.183,E2 -15474.183} C_VEL
LIN {X 0,Y 311.575,Z 393.986,A -85,B 0,C 180,E1 -15475.798,E2 -15475.798} C_VEL
LIN {X 0,Y 311.38,Z 398.748,A -85,B 0,C 180,E1 -15477.414,E2 -15477.414} C_VEL
LIN {X 0,Y 311.359,Z 402.843,A -85,B 0,C 180,E1 -15479.355,E2 -15479.355} C_VEL
LIN {X 0,Y 311.562,Z 405.41,A -85,B 0,C 180,E1 -15481.294,E2 -15481.294} C_VEL
LIN {X 0,Y 311.814,Z 406.321,A -85,B 0,C 180,E1 -15482.585,E2 -15482.585} C_VEL
LIN {X 0,Y 312.172,Z 406.606,A -85,B 0,C 180,E1 -15483.874,E2 -15483.874} C_VEL
LIN {X 0,Y 312.766,Z 406.254,A -85,B 0,C 180,E1 -15485.158,E2 -15485.158} C_VEL
LIN {X 0,Y 313.485,Z 405.297,A -85,B 0,C 180,E1 -15486.438,E2 -15486.438} C_VEL
LIN {X 0,Y 314.839,Z 402.658,A -85,B 0,C 180,E1 -15488.344,E2 -15488.344} C_VEL
LIN {X 0,Y 316.378,Z 398.521,A -85,B 0,C 180,E1 -15490.238,E2 -15490.238} C_VEL
LIN {X 0,Y 318.166,Z 392.757,A -85,B 0,C 180,E1 -15492.115,E2 -15492.115} C_VEL
LIN {X 0,Y 320.009,Z 386.463,A -85,B 0,C 180,E1 -15493.657,E2 -15493.657} C_VEL
LIN {X 0,Y 322.018,Z 378.526,A -85,B 0,C 180,E1 -15495.184,E2 -15495.184} C_VEL
LIN {X 0,Y 322.792,Z 373.469,A -85,B 0,C 180,E1 -15496.036,E2 -15496.036} C_VEL
LIN {X 0,Y 321.955,Z 366.05,A -85,B 0,C 180,E1 -15497.403,E2 -15497.403} C_VEL
LIN {X 0,Y 319.705,Z 356.786,A -85,B 0,C 180,E1 -15499.045,E2 -15499.045} C_VEL
LIN {X 0,Y 316.99,Z 348.765,A -85,B 0,C 180,E1 -15500.468,E2 -15500.468} C_VEL
LIN {X 0,Y 315.246,Z 344.172,A -85,B 0,C 180,E1 -15501.284,E2 -15501.284} C_VEL
LIN {X 0,Y 316.246,Z 340.325,A -85,B 0,C 180,E1 -15504.978,E2 -15504.978} C_VEL
LIN {X 0,Y 317.088,Z 337.757,A -85,B 0,C 180,E1 -15507.741,E2 -15507.741} C_VEL
LIN {X 0,Y 317.951,Z 335.517,A -85,B 0,C 180,E1 -15510.558,E2 -15510.558} C_VEL
LIN {X 0,Y 318.451,Z 333.783,A -85,B 0,C 180,E1 -15513.488,E2 -15513.488} C_VEL
LIN {X 0,Y 318.623,Z 333.031,A -85,B 0,C 180,E1 -15515.301,E2 -15515.301} C_VEL
LIN {X 0,Y 318.783,Z 332.407,A -85,B 0,C 180,E1 -15518.121,E2 -15518.121} C_VEL
LIN {X 0,Y 319.023,Z 332.42,A -85,B 0,C 180,E1 -15521.495,E2 -15521.495} C_VEL
LIN {X 0,Y 319.415,Z 333.311,A -85,B 0,C 180,E1 -15524.758,E2 -15524.758} C_VEL
LIN {X 0,Y 319.993,Z 335.372,A -85,B 0,C 180,E1 -15528.311,E2 -15528.311} C_VEL
LIN {X 0,Y 320.463,Z 337.245,A -85,B 0,C 180,E1 -15530.506,E2 -15530.506} C_VEL
LIN {X 0,Y 321.224,Z 340.883,A -85,B 0,C 180,E1 -15533.791,E2 -15533.791} C_VEL
LIN {X 0,Y 322.132,Z 345.389,A -85,B 0,C 180,E1 -15536.946,E2 -15536.946} C_VEL
LIN {X 0,Y 322.217,Z 346.638,A -85,B 0,C 180,E1 -15537.699,E2 -15537.699} C_VEL
LIN {X 0,Y 321.452,Z 349.439,A -85,B 0,C 180,E1 -15539.083,E2 -15539.083} C_VEL
LIN {X 0,Y 318.226,Z 358.674,A -85,B 0,C 180,E1 -15543.08,E2 -15543.08} C_VEL
LIN {X 0,Y 317.735,Z 360.615,A -85,B 0,C 180,E1 -15543.824,E2 -15543.824} C_VEL
LIN {X 0,Y 320.432,Z 372.097,A -85,B 0,C 180,E1 -15545.025,E2 -15545.025} C_VEL
LIN {X 0,Y 322.174,Z 384.906,A -85,B 0,C 180,E1 -15546.38,E2 -15546.38} C_VEL
LIN {X 0,Y 322.387,Z 395.167,A -85,B 0,C 180,E1 -15547.516,E2 -15547.516} C_VEL
LIN {X 0,Y 321.271,Z 406.355,A -85,B 0,C 180,E1 -15548.841,E2 -15548.841} C_VEL
LIN {X 0,Y 318.893,Z 417.429,A -85,B 0,C 180,E1 -15550.361,E2 -15550.361} C_VEL
LIN {X 0,Y 316.853,Z 426.503,A -85,B 0,C 180,E1 -15551.909,E2 -15551.909} C_VEL
LIN {X 0,Y 314.956,Z 435.127,A -85,B 0,C 180,E1 -15553.736,E2 -15553.736} C_VEL
LIN {X 0,Y 313.384,Z 442.649,A -85,B 0,C 180,E1 -15555.718,E2 -15555.718} C_VEL
LIN {X 0,Y 312.203,Z 448.541,A -85,B 0,C 180,E1 -15557.652,E2 -15557.652} C_VEL
LIN {X 0,Y 311.454,Z 453.222,A -85,B 0,C 180,E1 -15559.6,E2 -15559.6} C_VEL
LIN {X 0,Y 311.103,Z 456.844,A -85,B 0,C 180,E1 -15561.556,E2 -15561.556} C_VEL
LIN {X 0,Y 311.027,Z 459.817,A -85,B 0,C 180,E1 -15563.852,E2 -15563.852} C_VEL
LIN {X 0,Y 311.124,Z 461.478,A -85,B 0,C 180,E1 -15566.114,E2 -15566.114} C_VEL
LIN {X 0,Y 311.337,Z 461.843,A -85,B 0,C 180,E1 -15567.412,E2 -15567.412} C_VEL
LIN {X 0,Y 311.51,Z 461.761,A -85,B 0,C 180,E1 -15568.707,E2 -15568.707} C_VEL
LIN {X 0,Y 311.493,Z 461.241,A -85,B 0,C 180,E1 -15570,E2 -15570} C_VEL
LIN {X 0,Y 311.559,Z 460.165,A -85,B 0,C 180,E1 -15571.454,E2 -15571.454} C_VEL
LIN {X 0,Y 311.464,Z 460.275,A -85,B 0,C 180,E1 -15572.587,E2 -15572.587} C_VEL
LIN {X 0,Y 311.225,Z 459.756,A -85,B 0,C 180,E1 -15573.885,E2 -15573.885} C_VEL
LIN {X 0,Y 311.184,Z 458.563,A -85,B 0,C 180,E1 -15575.183,E2 -15575.183} C_VEL
LIN {X 0,Y 311.228,Z 456.678,A -85,B 0,C 180,E1 -15576.483,E2 -15576.483} C_VEL
LIN {X 0,Y 311.289,Z 454.057,A -85,B 0,C 180,E1 -15577.785,E2 -15577.785} C_VEL
LIN {X 0,Y 311.579,Z 448.592,A -85,B 0,C 180,E1 -15579.74,E2 -15579.74} C_VEL
LIN {X 0,Y 312.022,Z 442.488,A -85,B 0,C 180,E1 -15581.367,E2 -15581.367} C_VEL
LIN {X 0,Y 312.599,Z 436.327,A -85,B 0,C 180,E1 -15582.662,E2 -15582.662} C_VEL
LIN {X 0,Y 313.27,Z 428.637,A -85,B 0,C 180,E1 -15583.956,E2 -15583.956} C_VEL
LIN {X 0,Y 313.929,Z 419.323,A -85,B 0,C 180,E1 -15585.195,E2 -15585.195} C_VEL
LIN {X 0,Y 314.423,Z 409.819,A -85,B 0,C 180,E1 -15586.158,E2 -15586.158} C_VEL
LIN {X 0,Y 314.931,Z 399.752,A -85,B 0,C 180,E1 -15586.906,E2 -15586.906} C_VEL
LIN {X 0,Y 314.231,Z 389.464,A -85,B 0,C 180,E1 -15587.574,E2 -15587.574} C_VEL
LIN {X 0,Y 314.678,Z 376.697,A -85,B 0,C 180,E1 -15589.234,E2 -15589.234} C_VEL
LIN {X 0,Y 315.242,Z 370.524,A -85,B 0,C 180,E1 -15590.079,E2 -15590.079} C_VEL
LIN {X 0,Y 314.733,Z 361.549,A -85,B 0,C 180,E1 -15591.62,E2 -15591.62} C_VEL
LIN {X 0,Y 314.56,Z 354.626,A -85,B 0,C 180,E1 -15592.928,E2 -15592.928} C_VEL
LIN {X 0,Y 314.625,Z 346.413,A -85,B 0,C 180,E1 -15594.673,E2 -15594.673} C_VEL
LIN {X 0,Y 316.429,Z 335.39,A -85,B 0,C 180,E1 -15598.524,E2 -15598.524} C_VEL
LIN {X 0,Y 317.397,Z 329.455,A -85,B 0,C 180,E1 -15600.616,E2 -15600.616} C_VEL
LIN {X 0,Y 315.335,Z 319.454,A -85,B 0,C 180,E1 -15604.447,E2 -15604.447} C_VEL
LIN {X 0,Y 314.96,Z 317.689,A -85,B 0,C 180,E1 -15605.184,E2 -15605.184} C_VEL
LIN {X 0,Y 315.107,Z 315.685,A -85,B 0,C 180,E1 -15607.027,E2 -15607.027} C_VEL
LIN {X 0,Y 315.507,Z 314.242,A -85,B 0,C 180,E1 -15608.771,E2 -15608.771} C_VEL
LIN {X 0,Y 315.53,Z 313.643,A -85,B 0,C 180,E1 -15610.771,E2 -15610.771} C_VEL
LIN {X 0,Y 315.606,Z 314.226,A -85,B 0,C 180,E1 -15614.553,E2 -15614.553} C_VEL
LIN {X 0,Y 315.941,Z 315.6,A -85,B 0,C 180,E1 -15617.229,E2 -15617.229} C_VEL
LIN {X 0,Y 316.678,Z 318.579,A -85,B 0,C 180,E1 -15620.964,E2 -15620.964} C_VEL
LIN {X 0,Y 317.282,Z 321.059,A -85,B 0,C 180,E1 -15623.267,E2 -15623.267} C_VEL
LIN {X 0,Y 317.871,Z 324.874,A -85,B 0,C 180,E1 -15626.443,E2 -15626.443} C_VEL
LIN {X 0,Y 318.211,Z 329.271,A -85,B 0,C 180,E1 -15629.469,E2 -15629.469} C_VEL
LIN {X 0,Y 317.329,Z 335.32,A -85,B 0,C 180,E1 -15632.997,E2 -15632.997} C_VEL
LIN {X 0,Y 316.45,Z 342.665,A -85,B 0,C 180,E1 -15637.128,E2 -15637.128} C_VEL
LIN {X 0,Y 315.743,Z 350.063,A -85,B 0,C 180,E1 -15641.169,E2 -15641.169} C_VEL
LIN {X 0,Y 315.534,Z 352.898,A -85,B 0,C 180,E1 -15642.688,E2 -15642.688} C_VEL
LIN {X 0,Y 318.764,Z 362.73,A -85,B 0,C 180,E1 -15643.935,E2 -15643.935} C_VEL
LIN {X 0,Y 320.294,Z 369.508,A -85,B 0,C 180,E1 -15644.899,E2 -15644.899} C_VEL
LIN {X 0,Y 320.542,Z 371.446,A -85,B 0,C 180,E1 -15645.173,E2 -15645.173} C_VEL
LIN {X 0,Y 319.21,Z 380.69,A -85,B 0,C 180,E1 -15646.47,E2 -15646.47} C_VEL
LIN {X 0,Y 317.984,Z 386.821,A -85,B 0,C 180,E1 -15647.554,E2 -15647.554} C_VEL
LIN {X 0,Y 316.626,Z 393.539,A -85,B 0,C 180,E1 -15649.123,E2 -15649.123} C_VEL
LIN {X 0,Y 315.674,Z 397.633,A -85,B 0,C 180,E1 -15650.386,E2 -15650.386} C_VEL
LIN {X 0,Y 314.299,Z 402.122,A -85,B 0,C 180,E1 -15652.288,E2 -15652.288} C_VEL
LIN {X 0,Y 313.483,Z 404.131,A -85,B 0,C 180,E1 -15653.562,E2 -15653.562} C_VEL
LIN {X 0,Y 312.762,Z 405.42,A -85,B 0,C 180,E1 -15654.842,E2 -15654.842} C_VEL
LIN {X 0,Y 312.146,Z 406.011,A -85,B 0,C 180,E1 -15656.125,E2 -15656.125} C_VEL
LIN {X 0,Y 311.794,Z 405.899,A -85,B 0,C 180,E1 -15657.415,E2 -15657.415} C_VEL
LIN {X 0,Y 311.547,Z 405.105,A -85,B 0,C 180,E1 -15658.706,E2 -15658.706} C_VEL
LIN {X 0,Y 311.336,Z 402.665,A -85,B 0,C 180,E1 -15660.645,E2 -15660.645} C_VEL
LIN {X 0,Y 311.371,Z 400.089,A -85,B 0,C 180,E1 -15661.939,E2 -15661.939} C_VEL
LIN {X 0,Y 311.459,Z 394.68,A -85,B 0,C 180,E1 -15663.88,E2 -15663.88} C_VEL
LIN {X 0,Y 311.805,Z 388.391,A -85,B 0,C 180,E1 -15665.495,E2 -15665.495} C_VEL
LIN {X 0,Y 311.998,Z 382.227,A -85,B 0,C 180,E1 -15666.745,E2 -15666.745} C_VEL
LIN {X 0,Y 312.186,Z 373.652,A -85,B 0,C 180,E1 -15668.086,E2 -15668.086} C_VEL
LIN {X 0,Y 312.402,Z 365.686,A -85,B 0,C 180,E1 -15669.059,E2 -15669.059} C_VEL
LIN {X 0,Y 312.674,Z 357.052,A -85,B 0,C 180,E1 -15669.867,E2 -15669.867} C_VEL
LIN {X 0,Y 312.437,Z 351.429,A -85,B 0,C 180,E1 -15670.283,E2 -15670.283} C_VEL
LIN {X 0,Y 311.913,Z 346.832,A -85,B 0,C 180,E1 -15670.588,E2 -15670.588} C_VEL
LIN {X 0,Y 312.023,Z 338.5,A -85,B 0,C 180,E1 -15674.411,E2 -15674.411} C_VEL
LIN {X 0,Y 312.09,Z 330.004,A -85,B 0,C 180,E1 -15678.375,E2 -15678.375} C_VEL
LIN {X 0,Y 312.244,Z 322.736,A -85,B 0,C 180,E1 -15681.799,E2 -15681.799} C_VEL
LIN {X 0,Y 312.43,Z 315.383,A -85,B 0,C 180,E1 -15685.3,E2 -15685.3} C_VEL
LIN {X 0,Y 312.601,Z 308.165,A -85,B 0,C 180,E1 -15688.74,E2 -15688.74} C_VEL
LIN {X 0,Y 312.705,Z 305.531,A -85,B 0,C 180,E1 -15690.002,E2 -15690.002} C_VEL
LIN {X 0,Y 312.501,Z 305.555,A -85,B 0,C 180,E1 -15694.208,E2 -15694.208} C_VEL
LIN {X 0,Y 312.508,Z 305.558,A -85,B 0,C 180,E1 -15697.385,E2 -15697.385} C_VEL
LIN {X 0,Y 312.434,Z 305.566,A -85,B 0,C 180,E1 -15700.715,E2 -15700.715} C_VEL
LIN {X 0,Y 312.444,Z 305.563,A -85,B 0,C 180,E1 -15704.208,E2 -15704.208} C_VEL
LIN {X 0,Y 312.476,Z 305.559,A -85,B 0,C 180,E1 -15707.917,E2 -15707.917} C_VEL
LIN {X 0,Y 312.498,Z 305.556,A -85,B 0,C 180,E1 -15711.916,E2 -15711.916} C_VEL
LIN {X 0,Y 312.524,Z 305.554,A -85,B 0,C 180,E1 -15714.219,E2 -15714.219} C_VEL
LIN {X 0,Y 312.495,Z 305.557,A -85,B 0,C 180,E1 -15717.333,E2 -15717.333} C_VEL
LIN {X 0,Y 312.543,Z 305.551,A -85,B 0,C 180,E1 -15721.275,E2 -15721.275} C_VEL
LIN {X 0,Y 312.575,Z 305.55,A -85,B 0,C 180,E1 -15724.71,E2 -15724.71} C_VEL
LIN {X 0,Y 312.577,Z 305.546,A -85,B 0,C 180,E1 -15727.528,E2 -15727.528} C_VEL
LIN {X 0,Y 312.628,Z 305.54,A -85,B 0,C 180,E1 -15731.656,E2 -15731.656} C_VEL
LIN {X 0,Y 312.682,Z 305.534,A -85,B 0,C 180,E1 -15735.686,E2 -15735.686} C_VEL
LIN {X 0,Y 312.674,Z 305.535,A -85,B 0,C 180,E1 -15739.641,E2 -15739.641} C_VEL
LIN {X 0,Y 312.785,Z 305.525,A -85,B 0,C 180,E1 -15742.252,E2 -15742.252} C_VEL
LIN {X 0,Y 312.679,Z 305.533,A -85,B 0,C 180,E1 -15744.842,E2 -15744.842} C_VEL
LIN {X 0,Y 312.954,Z 305.5,A -85,B 0,C 180,E1 -15748.713,E2 -15748.713} C_VEL
LIN {X 0,Y 312.894,Z 305.507,A -85,B 0,C 180,E1 -15752.575,E2 -15752.575} C_VEL
LIN {X 0,Y 312.83,Z 305.515,A -85,B 0,C 180,E1 -15756.45,E2 -15756.45} C_VEL
LIN {X 0,Y 312.739,Z 305.526,A -85,B 0,C 180,E1 -15759.051,E2 -15759.051} C_VEL
LIN {X 0,Y 312.622,Z 305.541,A -85,B 0,C 180,E1 -15762.992,E2 -15762.992} C_VEL
LIN {X 0,Y 312.627,Z 305.545,A -85,B 0,C 180,E1 -15765.65,E2 -15765.65} C_VEL
LIN {X 0,Y 312.62,Z 305.543,A -85,B 0,C 180,E1 -15769.238,E2 -15769.238} C_VEL
LIN {X 0,Y 312.535,Z 305.552,A -85,B 0,C 180,E1 -15772.79,E2 -15772.79} C_VEL
LIN {X 0,Y 312.593,Z 305.545,A -85,B 0,C 180,E1 -15775.937,E2 -15775.937} C_VEL
LIN {X 0,Y 312.536,Z 305.554,A -85,B 0,C 180,E1 -15779.651,E2 -15779.651} C_VEL
LIN {X 0,Y 312.51,Z 305.556,A -85,B 0,C 180,E1 -15783.69,E2 -15783.69} C_VEL
LIN {X 0,Y 312.518,Z 305.557,A -85,B 0,C 180,E1 -15787.386,E2 -15787.386} C_VEL
LIN {X 0,Y 312.482,Z 305.56,A -85,B 0,C 180,E1 -15790.711,E2 -15790.711} C_VEL
LIN {X 0,Y 312.444,Z 305.563,A -85,B 0,C 180,E1 -15794.211,E2 -15794.211} C_VEL
LIN {X 0,Y 312.448,Z 305.562,A -85,B 0,C 180,E1 -15797.926,E2 -15797.926} C_VEL
LIN {X 0,Y 312.477,Z 305.559,A -85,B 0,C 180,E1 -15801.924,E2 -15801.924} C_VEL
LIN {X 0,Y 312.525,Z 305.553,A -85,B 0,C 180,E1 -15804.222,E2 -15804.222} C_VEL
LIN {X 0,Y 312.715,Z 305.636,A -85,B 0,C 180,E1 -15808.385,E2 -15808.385} C_VEL
LIN {X 0,Y 312.861,Z 308.671,A -85,B 0,C 180,E1 -15810.385,E2 -15810.385} C_VEL
LIN {X 0,Y 312.395,Z 314.57,A -85,B 0,C 180,E1 -15814.144,E2 -15814.144} C_VEL
LIN {X 0,Y 312.011,Z 321.037,A -85,B 0,C 180,E1 -15818.184,E2 -15818.184} C_VEL
LIN {X 0,Y 311.734,Z 326.624,A -85,B 0,C 180,E1 -15821.603,E2 -15821.603} C_VEL
LIN {X 0,Y 311.488,Z 333.334,A -85,B 0,C 180,E1 -15825.631,E2 -15825.631} C_VEL
LIN {X 0,Y 311.397,Z 336.922,A -85,B 0,C 180,E1 -15827.745,E2 -15827.745} C_VEL
LIN {X 0,Y 312.621,Z 349.263,A -85,B 0,C 180,E1 -15828.657,E2 -15828.657} C_VEL
LIN {X 0,Y 313.306,Z 354.878,A -85,B 0,C 180,E1 -15829.174,E2 -15829.174} C_VEL
LIN {X 0,Y 312.97,Z 362.174,A -85,B 0,C 180,E1 -15829.95,E2 -15829.95} C_VEL
LIN {X 0,Y 312.005,Z 367.055,A -85,B 0,C 180,E1 -15830.538,E2 -15830.538} C_VEL
LIN {X 0,Y 308.81,Z 374.568,A -85,B 0,C 180,E1 -15831.581,E2 -15831.581} C_VEL
LIN {X 0,Y 305.725,Z 381.5,A -85,B 0,C 180,E1 -15832.772,E2 -15832.772} C_VEL
LIN {X 0,Y 304.942,Z 385.47,A -85,B 0,C 180,E1 -15833.582,E2 -15833.582} C_VEL
LIN {X 0,Y 304.605,Z 391.534,A -85,B 0,C 180,E1 -15835.038,E2 -15835.038} C_VEL
LIN {X 0,Y 304.341,Z 396.969,A -85,B 0,C 180,E1 -15836.692,E2 -15836.692} C_VEL
LIN {X 0,Y 304.29,Z 401.853,A -85,B 0,C 180,E1 -15838.678,E2 -15838.678} C_VEL
LIN {X 0,Y 304.341,Z 404.218,A -85,B 0,C 180,E1 -15840.002,E2 -15840.002} C_VEL
LIN {X 0,Y 304.491,Z 405.923,A -85,B 0,C 180,E1 -15841.324,E2 -15841.324} C_VEL
LIN {X 0,Y 304.78,Z 406.989,A -85,B 0,C 180,E1 -15842.645,E2 -15842.645} C_VEL
LIN {X 0,Y 305.149,Z 407.434,A -85,B 0,C 180,E1 -15843.964,E2 -15843.964} C_VEL
LIN {X 0,Y 305.764,Z 407.234,A -85,B 0,C 180,E1 -15845.277,E2 -15845.277} C_VEL
LIN {X 0,Y 306.518,Z 406.414,A -85,B 0,C 180,E1 -15846.585,E2 -15846.585} C_VEL
LIN {X 0,Y 307.937,Z 404.009,A -85,B 0,C 180,E1 -15848.533,E2 -15848.533} C_VEL
LIN {X 0,Y 309.587,Z 400.178,A -85,B 0,C 180,E1 -15850.465,E2 -15850.465} C_VEL
LIN {X 0,Y 311.491,Z 394.772,A -85,B 0,C 180,E1 -15852.379,E2 -15852.379} C_VEL
LIN {X 0,Y 313.386,Z 388.832,A -85,B 0,C 180,E1 -15853.952,E2 -15853.952} C_VEL
LIN {X 0,Y 315.488,Z 381.383,A -85,B 0,C 180,E1 -15855.506,E2 -15855.506} C_VEL
LIN {X 0,Y 316.635,Z 376.073,A -85,B 0,C 180,E1 -15856.456,E2 -15856.456} C_VEL
LIN {X 0,Y 316.002,Z 369.172,A -85,B 0,C 180,E1 -15857.808,E2 -15857.808} C_VEL
LIN {X 0,Y 313.962,Z 359.757,A -85,B 0,C 180,E1 -15859.621,E2 -15859.621} C_VEL
LIN {X 0,Y 310.236,Z 348.717,A -85,B 0,C 180,E1 -15861.75,E2 -15861.75} C_VEL
LIN {X 0,Y 308.721,Z 344.988,A -85,B 0,C 180,E1 -15862.477,E2 -15862.477} C_VEL
LIN {X 0,Y 309.585,Z 341.871,A -85,B 0,C 180,E1 -15865.553,E2 -15865.553} C_VEL
LIN {X 0,Y 310.491,Z 339.423,A -85,B 0,C 180,E1 -15868.383,E2 -15868.383} C_VEL
LIN {X 0,Y 311.344,Z 337.364,A -85,B 0,C 180,E1 -15871.279,E2 -15871.279} C_VEL
LIN {X 0,Y 311.846,Z 335.826,A -85,B 0,C 180,E1 -15874.294,E2 -15874.294} C_VEL
LIN {X 0,Y 312.083,Z 334.975,A -85,B 0,C 180,E1 -15877.449,E2 -15877.449} C_VEL
LIN {X 0,Y 312.297,Z 334.872,A -85,B 0,C 180,E1 -15880.741,E2 -15880.741} C_VEL
LIN {X 0,Y 312.697,Z 335.679,A -85,B 0,C 180,E1 -15884.168,E2 -15884.168} C_VEL
LIN {X 0,Y 313.273,Z 337.582,A -85,B 0,C 180,E1 -15887.761,E2 -15887.761} C_VEL
LIN {X 0,Y 313.965,Z 340.468,A -85,B 0,C 180,E1 -15891.187,E2 -15891.187} C_VEL
LIN {X 0,Y 314.77,Z 344.325,A -85,B 0,C 180,E1 -15894.513,E2 -15894.513} C_VEL
LIN {X 0,Y 315.425,Z 347.747,A -85,B 0,C 180,E1 -15896.915,E2 -15896.915} C_VEL
LIN {X 0,Y 315.378,Z 349.343,A -85,B 0,C 180,E1 -15897.868,E2 -15897.868} C_VEL
LIN {X 0,Y 313.944,Z 353.272,A -85,B 0,C 180,E1 -15899.756,E2 -15899.756} C_VEL
LIN {X 0,Y 311.552,Z 360.154,A -85,B 0,C 180,E1 -15902.728,E2 -15902.728} C_VEL
LIN {X 0,Y 314.462,Z 372.685,A -85,B 0,C 180,E1 -15904.162,E2 -15904.162} C_VEL
LIN {X 0,Y 316.012,Z 384.644,A -85,B 0,C 180,E1 -15905.528,E2 -15905.528} C_VEL
LIN {X 0,Y 316.298,Z 395.166,A -85,B 0,C 180,E1 -15906.776,E2 -15906.776} C_VEL
LIN {X 0,Y 315.211,Z 405.622,A -85,B 0,C 180,E1 -15908.071,E2 -15908.071} C_VEL
LIN {X 0,Y 312.772,Z 416.592,A -85,B 0,C 180,E1 -15909.617,E2 -15909.617} C_VEL
LIN {X 0,Y 310.584,Z 425.621,A -85,B 0,C 180,E1 -15911.189,E2 -15911.189} C_VEL
LIN {X 0,Y 308.714,Z 433.163,A -85,B 0,C 180,E1 -15912.785,E2 -15912.785} C_VEL
LIN {X 0,Y 306.903,Z 440.612,A -85,B 0,C 180,E1 -15914.731,E2 -15914.731} C_VEL
LIN {X 0,Y 305.657,Z 446.702,A -85,B 0,C 180,E1 -15916.707,E2 -15916.707} C_VEL
LIN {X 0,Y 304.601,Z 451.592,A -85,B 0,C 180,E1 -15918.69,E2 -15918.69} C_VEL
LIN {X 0,Y 304.13,Z 455.409,A -85,B 0,C 180,E1 -15920.691,E2 -15920.691} C_VEL
LIN {X 0,Y 303.98,Z 457.386,A -85,B 0,C 180,E1 -15922.026,E2 -15922.026} C_VEL
LIN {X 0,Y 303.995,Z 460.072,A -85,B 0,C 180,E1 -15924.694,E2 -15924.694} C_VEL
LIN {X 0,Y 304.044,Z 460.773,A -85,B 0,C 180,E1 -15926.024,E2 -15926.024} C_VEL
LIN {X 0,Y 304.269,Z 461.05,A -85,B 0,C 180,E1 -15927.352,E2 -15927.352} C_VEL
LIN {X 0,Y 304.462,Z 460.912,A -85,B 0,C 180,E1 -15928.677,E2 -15928.677} C_VEL
LIN {X 0,Y 304.455,Z 460.296,A -85,B 0,C 180,E1 -15930,E2 -15930} C_VEL
LIN {X 0,Y 304.527,Z 459.256,A -85,B 0,C 180,E1 -15931.488,E2 -15931.488} C_VEL
LIN {X 0,Y 304.388,Z 459.485,A -85,B 0,C 180,E1 -15932.647,E2 -15932.647} C_VEL
LIN {X 0,Y 304.138,Z 459.099,A -85,B 0,C 180,E1 -15933.975,E2 -15933.975} C_VEL
LIN {X 0,Y 304.104,Z 458.045,A -85,B 0,C 180,E1 -15935.304,E2 -15935.304} C_VEL
LIN {X 0,Y 304.163,Z 455.172,A -85,B 0,C 180,E1 -15937.301,E2 -15937.301} C_VEL
LIN {X 0,Y 304.422,Z 450.681,A -85,B 0,C 180,E1 -15939.3,E2 -15939.3} C_VEL
LIN {X 0,Y 304.834,Z 445.452,A -85,B 0,C 180,E1 -15940.965,E2 -15940.965} C_VEL
LIN {X 0,Y 305.542,Z 438.733,A -85,B 0,C 180,E1 -15942.622,E2 -15942.622} C_VEL
LIN {X 0,Y 306.262,Z 431.884,A -85,B 0,C 180,E1 -15943.943,E2 -15943.943} C_VEL
LIN {X 0,Y 307.066,Z 423.328,A -85,B 0,C 180,E1 -15945.272,E2 -15945.272} C_VEL
LIN {X 0,Y 307.784,Z 414.593,A -85,B 0,C 180,E1 -15946.312,E2 -15946.312} C_VEL
LIN {X 0,Y 308.508,Z 404.7,A -85,B 0,C 180,E1 -15947.226,E2 -15947.226} C_VEL
LIN {X 0,Y 308.657,Z 396.867,A -85,B 0,C 180,E1 -15947.795,E2 -15947.795} C_VEL
LIN {X 0,Y 307.92,Z 388.685,A -85,B 0,C 180,E1 -15948.376,E2 -15948.376} C_VEL
LIN {X 0,Y 308.498,Z 378.207,A -85,B 0,C 180,E1 -15949.808,E2 -15949.808} C_VEL
LIN {X 0,Y 309.041,Z 372.101,A -85,B 0,C 180,E1 -15950.691,E2 -15950.691} C_VEL
LIN {X 0,Y 308.71,Z 359.434,A -85,B 0,C 180,E1 -15953.012,E2 -15953.012} C_VEL
LIN {X 0,Y 308.686,Z 348.968,A -85,B 0,C 180,E1 -15955.27,E2 -15955.27} C_VEL
LIN {X 0,Y 309.145,Z 338.546,A -85,B 0,C 180,E1 -15957.962,E2 -15957.962} C_VEL
LIN {X 0,Y 309.669,Z 334.419,A -85,B 0,C 180,E1 -15959.206,E2 -15959.206} C_VEL
LIN {X 0,Y 310.355,Z 330.503,A -85,B 0,C 180,E1 -15960.624,E2 -15960.624} C_VEL
LIN {X 0,Y 309.983,Z 328.436,A -85,B 0,C 180,E1 -15961.431,E2 -15961.431} C_VEL
LIN {X 0,Y 309.421,Z 322.369,A -85,B 0,C 180,E1 -15965.144,E2 -15965.144} C_VEL
LIN {X 0,Y 309.659,Z 319.493,A -85,B 0,C 180,E1 -15967.792,E2 -15967.792} C_VEL
LIN {X 0,Y 309.921,Z 318.274,A -85,B 0,C 180,E1 -15969.553,E2 -15969.553} C_VEL
LIN {X 0,Y 309.782,Z 317.883,A -85,B 0,C 180,E1 -15971.523,E2 -15971.523} C_VEL
LIN {X 0,Y 309.795,Z 318.529,A -85,B 0,C 180,E1 -15975.309,E2 -15975.309} C_VEL
LIN {X 0,Y 310.095,Z 320.218,A -85,B 0,C 180,E1 -15978.41,E2 -15978.41} C_VEL
LIN {X 0,Y 310.5,Z 321.956,A -85,B 0,C 180,E1 -15980.67,E2 -15980.67} C_VEL
LIN {X 0,Y 310.812,Z 323.498,A -85,B 0,C 180,E1 -15982.371,E2 -15982.371} C_VEL
LIN {X 0,Y 311.257,Z 325.828,A -85,B 0,C 180,E1 -15984.377,E2 -15984.377} C_VEL
LIN {X 0,Y 311.618,Z 329.17,A -85,B 0,C 180,E1 -15987.228,E2 -15987.228} C_VEL
LIN {X 0,Y 311.764,Z 332.08,A -85,B 0,C 180,E1 -15989.317,E2 -15989.317} C_VEL
LIN {X 0,Y 311.006,Z 336.766,A -85,B 0,C 180,E1 -15992.144,E2 -15992.144} C_VEL
LIN {X 0,Y 310.043,Z 343.234,A -85,B 0,C 180,E1 -15995.918,E2 -15995.918} C_VEL
LIN {X 0,Y 309.229,Z 350.595,A -85,B 0,C 180,E1 -16000.066,E2 -16000.066} C_VEL
LIN {X 0,Y 308.97,Z 353.955,A -85,B 0,C 180,E1 -16001.873,E2 -16001.873} C_VEL
LIN {X 0,Y 312.069,Z 363.127,A -85,B 0,C 180,E1 -16003.126,E2 -16003.126} C_VEL
LIN {X 0,Y 314.047,Z 371.733,A -85,B 0,C 180,E1 -16004.421,E2 -16004.421} C_VEL
LIN {X 0,Y 314.081,Z 374.737,A -85,B 0,C 180,E1 -16004.861,E2 -16004.861} C_VEL
LIN {X 0,Y 312.796,Z 382.518,A -85,B 0,C 180,E1 -16006.021,E2 -16006.021} C_VEL
LIN {X 0,Y 311.321,Z 389.075,A -85,B 0,C 180,E1 -16007.283,E2 -16007.283} C_VEL
LIN {X 0,Y 309.883,Z 395.382,A -85,B 0,C 180,E1 -16008.884,E2 -16008.884} C_VEL
LIN {X 0,Y 308.332,Z 400.893,A -85,B 0,C 180,E1 -16010.817,E2 -16010.817} C_VEL
LIN {X 0,Y 307.418,Z 403.464,A -85,B 0,C 180,E1 -16012.114,E2 -16012.114} C_VEL
LIN {X 0,Y 306.52,Z 405.283,A -85,B 0,C 180,E1 -16013.415,E2 -16013.415} C_VEL
LIN {X 0,Y 305.758,Z 406.394,A -85,B 0,C 180,E1 -16014.723,E2 -16014.723} C_VEL
LIN {X 0,Y 305.125,Z 406.821,A -85,B 0,C 180,E1 -16016.036,E2 -16016.036} C_VEL
LIN {X 0,Y 304.743,Z 406.558,A -85,B 0,C 180,E1 -16017.355,E2 -16017.355} C_VEL
LIN {X 0,Y 304.477,Z 405.621,A -85,B 0,C 180,E1 -16018.676,E2 -16018.676} C_VEL
LIN {X 0,Y 304.264,Z 402.925,A -85,B 0,C 180,E1 -16020.66,E2 -16020.66} C_VEL
LIN {X 0,Y 304.269,Z 398.514,A -85,B 0,C 180,E1 -16022.646,E2 -16022.646} C_VEL
LIN {X 0,Y 304.464,Z 393.263,A -85,B 0,C 180,E1 -16024.301,E2 -16024.301} C_VEL
LIN {X 0,Y 304.807,Z 386.38,A -85,B 0,C 180,E1 -16025.954,E2 -16025.954} C_VEL
LIN {X 0,Y 304.946,Z 378.716,A -85,B 0,C 180,E1 -16027.362,E2 -16027.362} C_VEL
LIN {X 0,Y 305.23,Z 369.874,A -85,B 0,C 180,E1 -16028.606,E2 -16028.606} C_VEL
LIN {X 0,Y 305.435,Z 360.568,A -85,B 0,C 180,E1 -16029.601,E2 -16029.601} C_VEL
LIN {X 0,Y 305.541,Z 353.375,A -85,B 0,C 180,E1 -16030.183,E2 -16030.183} C_VEL
LIN {X 0,Y 304.838,Z 347.451,A -85,B 0,C 180,E1 -16030.585,E2 -16030.585} C_VEL
LIN {X 0,Y 304.958,Z 338.873,A -85,B 0,C 180,E1 -16034.55,E2 -16034.55} C_VEL
LIN {X 0,Y 305.042,Z 329.818,A -85,B 0,C 180,E1 -16038.815,E2 -16038.815} C_VEL
LIN {X 0,Y 305.18,Z 322.55,A -85,B 0,C 180,E1 -16042.272,E2 -16042.272} C_VEL
LIN {X 0,Y 305.427,Z 314.392,A -85,B 0,C 180,E1 -16046.18,E2 -16046.18} C_VEL
LIN {X 0,Y 305.678,Z 306.406,A -85,B 0,C 180,E1 -16050.065,E2 -16050.065} C_VEL
LIN {X 0,Y 305.456,Z 306.437,A -85,B 0,C 180,E1 -16055.111,E2 -16055.111} C_VEL
LIN {X 0,Y 305.427,Z 306.438,A -85,B 0,C 180,E1 -16058.523,E2 -16058.523} C_VEL
LIN {X 0,Y 305.428,Z 306.438,A -85,B 0,C 180,E1 -16062.58,E2 -16062.58} C_VEL
LIN {X 0,Y 305.418,Z 306.439,A -85,B 0,C 180,E1 -16066.343,E2 -16066.343} C_VEL
LIN {X 0,Y 305.45,Z 306.434,A -85,B 0,C 180,E1 -16069.891,E2 -16069.891} C_VEL
LIN {X 0,Y 305.473,Z 306.431,A -85,B 0,C 180,E1 -16073.63,E2 -16073.63} C_VEL
LIN {X 0,Y 305.456,Z 306.436,A -85,B 0,C 180,E1 -16076.482,E2 -16076.482} C_VEL
LIN {X 0,Y 305.486,Z 306.432,A -85,B 0,C 180,E1 -16080.949,E2 -16080.949} C_VEL
LIN {X 0,Y 305.561,Z 306.422,A -85,B 0,C 180,E1 -16084.087,E2 -16084.087} C_VEL
LIN {X 0,Y 305.516,Z 306.43,A -85,B 0,C 180,E1 -16088.404,E2 -16088.404} C_VEL
LIN {X 0,Y 305.579,Z 306.418,A -85,B 0,C 180,E1 -16091.217,E2 -16091.217} C_VEL
LIN {X 0,Y 305.638,Z 306.41,A -85,B 0,C 180,E1 -16095.348,E2 -16095.348} C_VEL
LIN {X 0,Y 305.612,Z 306.414,A -85,B 0,C 180,E1 -16099.399,E2 -16099.399} C_VEL
LIN {X 0,Y 305.735,Z 306.403,A -85,B 0,C 180,E1 -16102.072,E2 -16102.072} C_VEL
LIN {X 0,Y 305.649,Z 306.409,A -85,B 0,C 180,E1 -16104.723,E2 -16104.723} C_VEL
LIN {X 0,Y 305.922,Z 306.376,A -85,B 0,C 180,E1 -16108.684,E2 -16108.684} C_VEL
LIN {X 0,Y 305.923,Z 306.376,A -85,B 0,C 180,E1 -16111.316,E2 -16111.316} C_VEL
LIN {X 0,Y 305.65,Z 306.409,A -85,B 0,C 180,E1 -16115.277,E2 -16115.277} C_VEL
LIN {X 0,Y 305.735,Z 306.403,A -85,B 0,C 180,E1 -16117.928,E2 -16117.928} C_VEL
LIN {X 0,Y 305.587,Z 306.42,A -85,B 0,C 180,E1 -16121.946,E2 -16121.946} C_VEL
LIN {X 0,Y 305.626,Z 306.413,A -85,B 0,C 180,E1 -16125.035,E2 -16125.035} C_VEL
LIN {X 0,Y 305.567,Z 306.424,A -85,B 0,C 180,E1 -16129.446,E2 -16129.446} C_VEL
LIN {X 0,Y 305.48,Z 306.432,A -85,B 0,C 180,E1 -16133.042,E2 -16133.042} C_VEL
LIN {X 0,Y 305.538,Z 306.423,A -85,B 0,C 180,E1 -16136.228,E2 -16136.228} C_VEL
LIN {X 0,Y 305.486,Z 306.432,A -85,B 0,C 180,E1 -16139.051,E2 -16139.051} C_VEL
LIN {X 0,Y 305.456,Z 306.436,A -85,B 0,C 180,E1 -16143.518,E2 -16143.518} C_VEL
LIN {X 0,Y 305.467,Z 306.433,A -85,B 0,C 180,E1 -16146.741,E2 -16146.741} C_VEL
LIN {X 0,Y 305.447,Z 306.435,A -85,B 0,C 180,E1 -16150.601,E2 -16150.601} C_VEL
LIN {X 0,Y 305.418,Z 306.439,A -85,B 0,C 180,E1 -16153.657,E2 -16153.657} C_VEL
LIN {X 0,Y 305.428,Z 306.438,A -85,B 0,C 180,E1 -16157.42,E2 -16157.42} C_VEL
LIN {X 0,Y 305.454,Z 306.434,A -85,B 0,C 180,E1 -16161.597,E2 -16161.597} C_VEL
LIN {X 0,Y 305.461,Z 306.436,A -85,B 0,C 180,E1 -16164.889,E2 -16164.889} C_VEL
LIN {X 0,Y 305.672,Z 306.456,A -85,B 0,C 180,E1 -16168.289,E2 -16168.289} C_VEL
LIN {X 0,Y 305.842,Z 308.455,A -85,B 0,C 180,E1 -16169.635,E2 -16169.635} C_VEL
LIN {X 0,Y 305.53,Z 313.002,A -85,B 0,C 180,E1 -16172.612,E2 -16172.612} C_VEL
LIN {X 0,Y 305.05,Z 319.778,A -85,B 0,C 180,E1 -16176.944,E2 -16176.944} C_VEL
LIN {X 0,Y 304.756,Z 325.517,A -85,B 0,C 180,E1 -16180.537,E2 -16180.537} C_VEL
LIN {X 0,Y 304.454,Z 332.166,A -85,B 0,C 180,E1 -16184.607,E2 -16184.607} C_VEL
LIN {X 0,Y 304.32,Z 337.255,A -85,B 0,C 180,E1 -16187.667,E2 -16187.667} C_VEL
LIN {X 0,Y 305.504,Z 349.244,A -85,B 0,C 180,E1 -16188.558,E2 -16188.558} C_VEL
LIN {X 0,Y 306.184,Z 356.552,A -85,B 0,C 180,E1 -16189.253,E2 -16189.253} C_VEL
LIN {X 0,Y 305.715,Z 366.54,A -85,B 0,C 180,E1 -16190.408,E2 -16190.408} C_VEL
LIN {X 0,Y 305.277,Z 375.987,A -85,B 0,C 180,E1 -16191.792,E2 -16191.792} C_VEL
LIN {X 0,Y 304.973,Z 384.564,A -85,B 0,C 180,E1 -16193.385,E2 -16193.385} C_VEL
LIN {X 0,Y 304.942,Z 385.47,A -85,B 0,C 180,E1 -16193.582,E2 -16193.582} C_VEL
LIN {X 0,Y 304.13,Z 389.193,A -85,B 0,C 180,E1 -16194.431,E2 -16194.431} C_VEL
LIN {X 0,Y 300.986,Z 394.601,A -85,B 0,C 180,E1 -16195.888,E2 -16195.888} C_VEL
LIN {X 0,Y 297.898,Z 399.269,A -85,B 0,C 180,E1 -16197.469,E2 -16197.469} C_VEL
LIN {X 0,Y 297.193,Z 401.713,A -85,B 0,C 180,E1 -16198.498,E2 -16198.498} C_VEL
LIN {X 0,Y 297.273,Z 404.567,A -85,B 0,C 180,E1 -16200.002,E2 -16200.002} C_VEL
LIN {X 0,Y 297.423,Z 406.412,A -85,B 0,C 180,E1 -16201.356,E2 -16201.356} C_VEL
LIN {X 0,Y 297.73,Z 407.616,A -85,B 0,C 180,E1 -16202.708,E2 -16202.708} C_VEL
LIN {X 0,Y 298.128,Z 408.198,A -85,B 0,C 180,E1 -16204.057,E2 -16204.057} C_VEL
LIN {X 0,Y 298.756,Z 408.16,A -85,B 0,C 180,E1 -16205.401,E2 -16205.401} C_VEL
LIN {X 0,Y 299.549,Z 407.509,A -85,B 0,C 180,E1 -16206.739,E2 -16206.739} C_VEL
LIN {X 0,Y 300.476,Z 406.269,A -85,B 0,C 180,E1 -16208.069,E2 -16208.069} C_VEL
LIN {X 0,Y 302.2,Z 403.197,A -85,B 0,C 180,E1 -16210.047,E2 -16210.047} C_VEL
LIN {X 0,Y 304.093,Z 398.639,A -85,B 0,C 180,E1 -16212.007,E2 -16212.007} C_VEL
LIN {X 0,Y 306.37,Z 392.432,A -85,B 0,C 180,E1 -16213.939,E2 -16213.939} C_VEL
LIN {X 0,Y 308.508,Z 385.755,A -85,B 0,C 180,E1 -16215.527,E2 -16215.527} C_VEL
LIN {X 0,Y 310.371,Z 379.131,A -85,B 0,C 180,E1 -16216.798,E2 -16216.798} C_VEL
LIN {X 0,Y 310.113,Z 372.658,A -85,B 0,C 180,E1 -16218.159,E2 -16218.159} C_VEL
LIN {X 0,Y 308.5,Z 363.839,A -85,B 0,C 180,E1 -16219.983,E2 -16219.983} C_VEL
LIN {X 0,Y 306.368,Z 356.451,A -85,B 0,C 180,E1 -16221.534,E2 -16221.534} C_VEL
LIN {X 0,Y 304.231,Z 350.667,A -85,B 0,C 180,E1 -16222.766,E2 -16222.766} C_VEL
LIN {X 0,Y 302.295,Z 345.529,A -85,B 0,C 180,E1 -16223.918,E2 -16223.918} C_VEL
LIN {X 0,Y 303.476,Z 342.291,A -85,B 0,C 180,E1 -16227.593,E2 -16227.593} C_VEL
LIN {X 0,Y 304.663,Z 339.612,A -85,B 0,C 180,E1 -16231.403,E2 -16231.403} C_VEL
LIN {X 0,Y 305.128,Z 338.362,A -85,B 0,C 180,E1 -16233.984,E2 -16233.984} C_VEL
LIN {X 0,Y 305.366,Z 337.575,A -85,B 0,C 180,E1 -16236.756,E2 -16236.756} C_VEL
LIN {X 0,Y 305.643,Z 337.366,A -85,B 0,C 180,E1 -16240.08,E2 -16240.08} C_VEL
LIN {X 0,Y 305.986,Z 338.06,A -85,B 0,C 180,E1 -16243.557,E2 -16243.557} C_VEL
LIN {X 0,Y 306.55,Z 339.796,A -85,B 0,C 180,E1 -16247.194,E2 -16247.194} C_VEL
LIN {X 0,Y 307.092,Z 342.038,A -85,B 0,C 180,E1 -16250.148,E2 -16250.148} C_VEL
LIN {X 0,Y 307.89,Z 345.663,A -85,B 0,C 180,E1 -16253.595,E2 -16253.595} C_VEL
LIN {X 0,Y 308.718,Z 350.094,A -85,B 0,C 180,E1 -16256.882,E2 -16256.882} C_VEL
LIN {X 0,Y 308.728,Z 350.912,A -85,B 0,C 180,E1 -16257.384,E2 -16257.384} C_VEL
LIN {X 0,Y 307.608,Z 354.178,A -85,B 0,C 180,E1 -16259.065,E2 -16259.065} C_VEL
LIN {X 0,Y 305.536,Z 359.64,A -85,B 0,C 180,E1 -16261.538,E2 -16261.538} C_VEL
LIN {X 0,Y 308.814,Z 374.518,A -85,B 0,C 180,E1 -16263.396,E2 -16263.396} C_VEL
LIN {X 0,Y 310.063,Z 385.641,A -85,B 0,C 180,E1 -16264.769,E2 -16264.769} C_VEL
LIN {X 0,Y 310.231,Z 396.275,A -85,B 0,C 180,E1 -16266.119,E2 -16266.119} C_VEL
LIN {X 0,Y 309.003,Z 406.25,A -85,B 0,C 180,E1 -16267.43,E2 -16267.43} C_VEL
LIN {X 0,Y 306.232,Z 417.849,A -85,B 0,C 180,E1 -16269.162,E2 -16269.162} C_VEL
LIN {X 0,Y 303.934,Z 426.438,A -85,B 0,C 180,E1 -16270.761,E2 -16270.761} C_VEL
LIN {X 0,Y 301.705,Z 434.708,A -85,B 0,C 180,E1 -16272.649,E2 -16272.649} C_VEL
LIN {X 0,Y 299.822,Z 441.94,A -85,B 0,C 180,E1 -16274.71,E2 -16274.71} C_VEL
LIN {X 0,Y 298.316,Z 448.406,A -85,B 0,C 180,E1 -16277.067,E2 -16277.067} C_VEL
LIN {X 0,Y 297.38,Z 452.745,A -85,B 0,C 180,E1 -16279.102,E2 -16279.102} C_VEL
LIN {X 0,Y 297.073,Z 455.06,A -85,B 0,C 180,E1 -16280.468,E2 -16280.468} C_VEL
LIN {X 0,Y 296.851,Z 458.397,A -85,B 0,C 180,E1 -16283.202,E2 -16283.202} C_VEL
LIN {X 0,Y 296.911,Z 459.437,A -85,B 0,C 180,E1 -16284.567,E2 -16284.567} C_VEL
LIN {X 0,Y 297.202,Z 460.253,A -85,B 0,C 180,E1 -16287.289,E2 -16287.289} C_VEL
LIN {X 0,Y 297.415,Z 460.026,A -85,B 0,C 180,E1 -16288.646,E2 -16288.646} C_VEL
LIN {X 0,Y 297.51,Z 458.254,A -85,B 0,C 180,E1 -16291.269,E2 -16291.269} C_VEL
LIN {X 0,Y 297.312,Z 458.69,A -85,B 0,C 180,E1 -16292.71,E2 -16292.71} C_VEL
LIN {X 0,Y 297.054,Z 458.441,A -85,B 0,C 180,E1 -16294.07,E2 -16294.07} C_VEL
LIN {X 0,Y 297.029,Z 457.53,A -85,B 0,C 180,E1 -16295.431,E2 -16295.431} C_VEL
LIN {X 0,Y 297.085,Z 454.944,A -85,B 0,C 180,E1 -16297.476,E2 -16297.476} C_VEL
LIN {X 0,Y 297.262,Z 452.308,A -85,B 0,C 180,E1 -16298.84,E2 -16298.84} C_VEL
LIN {X 0,Y 297.745,Z 446.87,A -85,B 0,C 180,E1 -16300.885,E2 -16300.885} C_VEL
LIN {X 0,Y 298.474,Z 440.835,A -85,B 0,C 180,E1 -16302.58,E2 -16302.58} C_VEL
LIN {X 0,Y 299.47,Z 433.064,A -85,B 0,C 180,E1 -16304.266,E2 -16304.266} C_VEL
LIN {X 0,Y 300.487,Z 424.129,A -85,B 0,C 180,E1 -16305.752,E2 -16305.752} C_VEL
LIN {X 0,Y 301.458,Z 414.805,A -85,B 0,C 180,E1 -16306.951,E2 -16306.951} C_VEL
LIN {X 0,Y 302.218,Z 406.567,A -85,B 0,C 180,E1 -16307.771,E2 -16307.771} C_VEL
LIN {X 0,Y 302.586,Z 398.101,A -85,B 0,C 180,E1 -16308.449,E2 -16308.449} C_VEL
LIN {X 0,Y 301.664,Z 388.303,A -85,B 0,C 180,E1 -16309.213,E2 -16309.213} C_VEL
LIN {X 0,Y 302.543,Z 378.491,A -85,B 0,C 180,E1 -16310.577,E2 -16310.577} C_VEL
LIN {X 0,Y 302.933,Z 374.988,A -85,B 0,C 180,E1 -16311.103,E2 -16311.103} C_VEL
LIN {X 0,Y 302.758,Z 362.53,A -85,B 0,C 180,E1 -16313.456,E2 -16313.456} C_VEL
LIN {X 0,Y 302.92,Z 352.057,A -85,B 0,C 180,E1 -16315.786,E2 -16315.786} C_VEL
LIN {X 0,Y 303.493,Z 342.343,A -85,B 0,C 180,E1 -16318.359,E2 -16318.359} C_VEL
LIN {X 0,Y 304.444,Z 335.498,A -85,B 0,C 180,E1 -16320.522,E2 -16320.522} C_VEL
LIN {X 0,Y 304.55,Z 333.334,A -85,B 0,C 180,E1 -16321.366,E2 -16321.366} C_VEL
LIN {X 0,Y 303.932,Z 326.754,A -85,B 0,C 180,E1 -16325.316,E2 -16325.316} C_VEL
LIN {X 0,Y 304.135,Z 323.302,A -85,B 0,C 180,E1 -16328.603,E2 -16328.603} C_VEL
LIN {X 0,Y 304.19,Z 322.379,A -85,B 0,C 180,E1 -16330.319,E2 -16330.319} C_VEL
LIN {X 0,Y 304.012,Z 322.157,A -85,B 0,C 180,E1 -16332.287,E2 -16332.287} C_VEL
LIN {X 0,Y 303.922,Z 322.258,A -85,B 0,C 180,E1 -16334.203,E2 -16334.203} C_VEL
LIN {X 0,Y 304.066,Z 323.674,A -85,B 0,C 180,E1 -16337.7,E2 -16337.7} C_VEL
LIN {X 0,Y 304.5,Z 326.281,A -85,B 0,C 180,E1 -16341.45,E2 -16341.45} C_VEL
LIN {X 0,Y 305.083,Z 329.764,A -85,B 0,C 180,E1 -16344.835,E2 -16344.835} C_VEL
LIN {X 0,Y 305.301,Z 332.459,A -85,B 0,C 180,E1 -16347.249,E2 -16347.249} C_VEL
LIN {X 0,Y 305.253,Z 335.656,A -85,B 0,C 180,E1 -16349.566,E2 -16349.566} C_VEL
LIN {X 0,Y 304.133,Z 341.545,A -85,B 0,C 180,E1 -16353.215,E2 -16353.215} C_VEL
LIN {X 0,Y 303.083,Z 348.778,A -85,B 0,C 180,E1 -16357.504,E2 -16357.504} C_VEL
LIN {X 0,Y 302.443,Z 354.997,A -85,B 0,C 180,E1 -16360.991,E2 -16360.991} C_VEL
LIN {X 0,Y 305.813,Z 364.701,A -85,B 0,C 180,E1 -16362.425,E2 -16362.425} C_VEL
LIN {X 0,Y 307.731,Z 373.28,A -85,B 0,C 180,E1 -16363.803,E2 -16363.803} C_VEL
LIN {X 0,Y 307.895,Z 376.119,A -85,B 0,C 180,E1 -16364.275,E2 -16364.275} C_VEL
LIN {X 0,Y 306.59,Z 383.404,A -85,B 0,C 180,E1 -16365.393,E2 -16365.393} C_VEL
LIN {X 0,Y 305.01,Z 389.963,A -85,B 0,C 180,E1 -16366.677,E2 -16366.677} C_VEL
LIN {X 0,Y 303.443,Z 396.269,A -85,B 0,C 180,E1 -16368.306,E2 -16368.306} C_VEL
LIN {X 0,Y 302.043,Z 400.901,A -85,B 0,C 180,E1 -16369.948,E2 -16369.948} C_VEL
LIN {X 0,Y 300.993,Z 403.691,A -85,B 0,C 180,E1 -16371.269,E2 -16371.269} C_VEL
LIN {X 0,Y 299.555,Z 406.411,A -85,B 0,C 180,E1 -16373.262,E2 -16373.262} C_VEL
LIN {X 0,Y 298.755,Z 407.367,A -85,B 0,C 180,E1 -16374.599,E2 -16374.599} C_VEL
LIN {X 0,Y 298.105,Z 407.637,A -85,B 0,C 180,E1 -16375.943,E2 -16375.943} C_VEL
LIN {X 0,Y 297.695,Z 407.215,A -85,B 0,C 180,E1 -16377.292,E2 -16377.292} C_VEL
LIN {X 0,Y 297.409,Z 406.12,A -85,B 0,C 180,E1 -16378.644,E2 -16378.644} C_VEL
LIN {X 0,Y 297.25,Z 404.337,A -85,B 0,C 180,E1 -16379.998,E2 -16379.998} C_VEL
LIN {X 0,Y 297.148,Z 401.819,A -85,B 0,C 180,E1 -16381.353,E2 -16381.353} C_VEL
LIN {X 0,Y 297.245,Z 396.444,A -85,B 0,C 180,E1 -16383.387,E2 -16383.387} C_VEL
LIN {X 0,Y 297.527,Z 390.271,A -85,B 0,C 180,E1 -16385.08,E2 -16385.08} C_VEL
LIN {X 0,Y 297.785,Z 383.988,A -85,B 0,C 180,E1 -16386.435,E2 -16386.435} C_VEL
LIN {X 0,Y 297.934,Z 376.256,A -85,B 0,C 180,E1 -16387.735,E2 -16387.735} C_VEL
LIN {X 0,Y 298.158,Z 368.234,A -85,B 0,C 180,E1 -16388.811,E2 -16388.811} C_VEL
LIN {X 0,Y 298.451,Z 358.085,A -85,B 0,C 180,E1 -16389.828,E2 -16389.828} C_VEL
LIN {X 0,Y 298.277,Z 352.466,A -85,B 0,C 180,E1 -16390.262,E2 -16390.262} C_VEL
LIN {X 0,Y 297.764,Z 348.047,A -85,B 0,C 180,E1 -16390.581,E2 -16390.581} C_VEL
LIN {X 0,Y 297.883,Z 340.338,A -85,B 0,C 180,E1 -16394.176,E2 -16394.176} C_VEL
LIN {X 0,Y 297.98,Z 331.063,A -85,B 0,C 180,E1 -16398.564,E2 -16398.564} C_VEL
LIN {X 0,Y 298.127,Z 323.59,A -85,B 0,C 180,E1 -16402.157,E2 -16402.157} C_VEL
LIN {X 0,Y 298.369,Z 316.088,A -85,B 0,C 180,E1 -16405.788,E2 -16405.788} C_VEL
LIN {X 0,Y 298.635,Z 307.283,A -85,B 0,C 180,E1 -16410.052,E2 -16410.052} C_VEL
LIN {X 0,Y 298.423,Z 307.309,A -85,B 0,C 180,E1 -16414.485,E2 -16414.485} C_VEL
LIN {X 0,Y 298.392,Z 307.314,A -85,B 0,C 180,E1 -16417.759,E2 -16417.759} C_VEL
LIN {X 0,Y 298.341,Z 307.323,A -85,B 0,C 180,E1 -16421.266,E2 -16421.266} C_VEL
LIN {X 0,Y 298.392,Z 307.318,A -85,B 0,C 180,E1 -16423.102,E2 -16423.102} C_VEL
LIN {X 0,Y 298.395,Z 307.318,A -85,B 0,C 180,E1 -16426.919,E2 -16426.919} C_VEL
LIN {X 0,Y 298.396,Z 307.316,A -85,B 0,C 180,E1 -16431.005,E2 -16431.005} C_VEL
LIN {X 0,Y 298.411,Z 307.311,A -85,B 0,C 180,E1 -16433.929,E2 -16433.929} C_VEL
LIN {X 0,Y 298.386,Z 307.314,A -85,B 0,C 180,E1 -16437.982,E2 -16437.982} C_VEL
LIN {X 0,Y 298.454,Z 307.306,A -85,B 0,C 180,E1 -16441.903,E2 -16441.903} C_VEL
LIN {X 0,Y 298.475,Z 307.305,A -85,B 0,C 180,E1 -16444.923,E2 -16444.923} C_VEL
LIN {X 0,Y 298.448,Z 307.306,A -85,B 0,C 180,E1 -16449.315,E2 -16449.315} C_VEL
LIN {X 0,Y 298.527,Z 307.3,A -85,B 0,C 180,E1 -16452.179,E2 -16452.179} C_VEL
LIN {X 0,Y 298.582,Z 307.29,A -85,B 0,C 180,E1 -16454.994,E2 -16454.994} C_VEL
LIN {X 0,Y 298.571,Z 307.291,A -85,B 0,C 180,E1 -16459.146,E2 -16459.146} C_VEL
LIN {X 0,Y 298.686,Z 307.279,A -85,B 0,C 180,E1 -16461.884,E2 -16461.884} C_VEL
LIN {X 0,Y 298.619,Z 307.286,A -85,B 0,C 180,E1 -16464.598,E2 -16464.598} C_VEL
LIN {X 0,Y 298.89,Z 307.252,A -85,B 0,C 180,E1 -16468.653,E2 -16468.653} C_VEL
LIN {X 0,Y 298.891,Z 307.252,A -85,B 0,C 180,E1 -16471.347,E2 -16471.347} C_VEL
LIN {X 0,Y 298.724,Z 307.272,A -85,B 0,C 180,E1 -16476.756,E2 -16476.756} C_VEL
LIN {X 0,Y 298.614,Z 307.288,A -85,B 0,C 180,E1 -16479.483,E2 -16479.483} C_VEL
LIN {X 0,Y 298.54,Z 307.298,A -85,B 0,C 180,E1 -16483.616,E2 -16483.616} C_VEL
LIN {X 0,Y 298.538,Z 307.295,A -85,B 0,C 180,E1 -16486.409,E2 -16486.409} C_VEL
LIN {X 0,Y 298.502,Z 307.303,A -85,B 0,C 180,E1 -16489.656,E2 -16489.656} C_VEL
LIN {X 0,Y 298.447,Z 307.31,A -85,B 0,C 180,E1 -16493.599,E2 -16493.599} C_VEL
LIN {X 0,Y 298.48,Z 307.302,A -85,B 0,C 180,E1 -16496.575,E2 -16496.575} C_VEL
LIN {X 0,Y 298.411,Z 307.313,A -85,B 0,C 180,E1 -16499.642,E2 -16499.642} C_VEL
LIN {X 0,Y 298.386,Z 307.315,A -85,B 0,C 180,E1 -16502.801,E2 -16502.801} C_VEL
LIN {X 0,Y 298.438,Z 307.309,A -85,B 0,C 180,E1 -16506.809,E2 -16506.809} C_VEL
LIN {X 0,Y 298.38,Z 307.32,A -85,B 0,C 180,E1 -16511.089,E2 -16511.089} C_VEL
LIN {X 0,Y 298.391,Z 307.318,A -85,B 0,C 180,E1 -16513.105,E2 -16513.105} C_VEL
LIN {X 0,Y 298.364,Z 307.321,A -85,B 0,C 180,E1 -16516.917,E2 -16516.917} C_VEL
LIN {X 0,Y 298.378,Z 307.319,A -85,B 0,C 180,E1 -16521.013,E2 -16521.013} C_VEL
LIN {X 0,Y 298.4,Z 307.312,A -85,B 0,C 180,E1 -16523.93,E2 -16523.93} C_VEL
LIN {X 0,Y 298.663,Z 307.406,A -85,B 0,C 180,E1 -16528.299,E2 -16528.299} C_VEL
LIN {X 0,Y 298.731,Z 310.686,A -85,B 0,C 180,E1 -16530.514,E2 -16530.514} C_VEL
LIN {X 0,Y 298.284,Z 316.3,A -85,B 0,C 180,E1 -16534.216,E2 -16534.216} C_VEL
LIN {X 0,Y 297.887,Z 321.9,A -85,B 0,C 180,E1 -16537.824,E2 -16537.824} C_VEL
LIN {X 0,Y 297.603,Z 327.653,A -85,B 0,C 180,E1 -16541.465,E2 -16541.465} C_VEL
LIN {X 0,Y 297.348,Z 334.497,A -85,B 0,C 180,E1 -16545.711,E2 -16545.711} C_VEL
LIN {X 0,Y 297.26,Z 337.775,A -85,B 0,C 180,E1 -16547.586,E2 -16547.586} C_VEL
LIN {X 0,Y 298.363,Z 349.209,A -85,B 0,C 180,E1 -16548.452,E2 -16548.452} C_VEL
LIN {X 0,Y 299.108,Z 356.615,A -85,B 0,C 180,E1 -16549.167,E2 -16549.167} C_VEL
LIN {X 0,Y 298.634,Z 366.701,A -85,B 0,C 180,E1 -16550.349,E2 -16550.349} C_VEL
LIN {X 0,Y 298.216,Z 375.798,A -85,B 0,C 180,E1 -16551.702,E2 -16551.702} C_VEL
LIN {X 0,Y 297.89,Z 383.982,A -85,B 0,C 180,E1 -16553.227,E2 -16553.227} C_VEL
LIN {X 0,Y 297.547,Z 391.208,A -85,B 0,C 180,E1 -16554.92,E2 -16554.92} C_VEL
LIN {X 0,Y 297.253,Z 396.912,A -85,B 0,C 180,E1 -16556.613,E2 -16556.613} C_VEL
LIN {X 0,Y 297.193,Z 401.713,A -85,B 0,C 180,E1 -16558.498,E2 -16558.498} C_VEL
LIN {X 0,Y 296.558,Z 403.927,A -85,B 0,C 180,E1 -16559.551,E2 -16559.551} C_VEL
LIN {X 0,Y 293.871,Z 406.824,A -85,B 0,C 180,E1 -16561.324,E2 -16561.324} C_VEL
LIN {X 0,Y 291.774,Z 408.319,A -85,B 0,C 180,E1 -16562.797,E2 -16562.797} C_VEL
LIN {X 0,Y 291.11,Z 408.894,A -85,B 0,C 180,E1 -16563.948,E2 -16563.948} C_VEL
LIN {X 0,Y 291.183,Z 408.966,A -85,B 0,C 180,E1 -16564.336,E2 -16564.336} C_VEL
LIN {X 0,Y 291.749,Z 409.086,A -85,B 0,C 180,E1 -16565.531,E2 -16565.531} C_VEL
LIN {X 0,Y 292.583,Z 408.6,A -85,B 0,C 180,E1 -16566.9,E2 -16566.9} C_VEL
LIN {X 0,Y 293.554,Z 407.515,A -85,B 0,C 180,E1 -16568.261,E2 -16568.261} C_VEL
LIN {X 0,Y 295.361,Z 404.714,A -85,B 0,C 180,E1 -16570.282,E2 -16570.282} C_VEL
LIN {X 0,Y 297.378,Z 400.523,A -85,B 0,C 180,E1 -16572.282,E2 -16572.282} C_VEL
LIN {X 0,Y 299.734,Z 394.715,A -85,B 0,C 180,E1 -16574.254,E2 -16574.254} C_VEL
LIN {X 0,Y 301.983,Z 388.421,A -85,B 0,C 180,E1 -16575.872,E2 -16575.872} C_VEL
LIN {X 0,Y 304.333,Z 380.716,A -85,B 0,C 180,E1 -16577.472,E2 -16577.472} C_VEL
LIN {X 0,Y 303.903,Z 373.329,A -85,B 0,C 180,E1 -16579.141,E2 -16579.141} C_VEL
LIN {X 0,Y 302.198,Z 364.243,A -85,B 0,C 180,E1 -16581.179,E2 -16581.179} C_VEL
LIN {X 0,Y 299.402,Z 355.199,A -85,B 0,C 180,E1 -16583.259,E2 -16583.259} C_VEL
LIN {X 0,Y 297.543,Z 350.311,A -85,B 0,C 180,E1 -16584.417,E2 -16584.417} C_VEL
LIN {X 0,Y 296.086,Z 346.845,A -85,B 0,C 180,E1 -16585.295,E2 -16585.295} C_VEL
LIN {X 0,Y 295.962,Z 346.315,A -85,B 0,C 180,E1 -16585.435,E2 -16585.435} C_VEL
LIN {X 0,Y 297.152,Z 343.541,A -85,B 0,C 180,E1 -16588.943,E2 -16588.943} C_VEL
LIN {X 0,Y 298.054,Z 341.697,A -85,B 0,C 180,E1 -16591.911,E2 -16591.911} C_VEL
LIN {X 0,Y 298.484,Z 340.618,A -85,B 0,C 180,E1 -16594.502,E2 -16594.502} C_VEL
LIN {X 0,Y 298.765,Z 339.976,A -85,B 0,C 180,E1 -16597.708,E2 -16597.708} C_VEL
LIN {X 0,Y 299.126,Z 340.087,A -85,B 0,C 180,E1 -16601.249,E2 -16601.249} C_VEL
LIN {X 0,Y 299.542,Z 341.105,A -85,B 0,C 180,E1 -16604.74,E2 -16604.74} C_VEL
LIN {X 0,Y 299.968,Z 342.408,A -85,B 0,C 180,E1 -16607.199,E2 -16607.199} C_VEL
LIN {X 0,Y 300.663,Z 345.267,A -85,B 0,C 180,E1 -16610.867,E2 -16610.867} C_VEL
LIN {X 0,Y 301.489,Z 349.477,A -85,B 0,C 180,E1 -16614.677,E2 -16614.677} C_VEL
LIN {X 0,Y 302.026,Z 352.531,A -85,B 0,C 180,E1 -16616.9,E2 -16616.9} C_VEL
LIN {X 0,Y 301.299,Z 355.138,A -85,B 0,C 180,E1 -16618.343,E2 -16618.343} C_VEL
LIN {X 0,Y 299.642,Z 359.15,A -85,B 0,C 180,E1 -16620.221,E2 -16620.221} C_VEL
LIN {X 0,Y 302.497,Z 372.01,A -85,B 0,C 180,E1 -16621.993,E2 -16621.993} C_VEL
LIN {X 0,Y 303.955,Z 382.327,A -85,B 0,C 180,E1 -16623.385,E2 -16623.385} C_VEL
LIN {X 0,Y 304.326,Z 394.377,A -85,B 0,C 180,E1 -16625.007,E2 -16625.007} C_VEL
LIN {X 0,Y 303.48,Z 403.53,A -85,B 0,C 180,E1 -16626.273,E2 -16626.273} C_VEL
LIN {X 0,Y 301.604,Z 412.332,A -85,B 0,C 180,E1 -16627.569,E2 -16627.569} C_VEL
LIN {X 0,Y 298.665,Z 422.544,A -85,B 0,C 180,E1 -16629.331,E2 -16629.331} C_VEL
LIN {X 0,Y 295.988,Z 431.623,A -85,B 0,C 180,E1 -16631.304,E2 -16631.304} C_VEL
LIN {X 0,Y 293.531,Z 440.084,A -85,B 0,C 180,E1 -16633.66,E2 -16633.66} C_VEL
LIN {X 0,Y 291.809,Z 446.745,A -85,B 0,C 180,E1 -16636.064,E2 -16636.064} C_VEL
LIN {X 0,Y 290.614,Z 451.232,A -85,B 0,C 180,E1 -16638.138,E2 -16638.138} C_VEL
LIN {X 0,Y 290.034,Z 454.695,A -85,B 0,C 180,E1 -16640.234,E2 -16640.234} C_VEL
LIN {X 0,Y 289.837,Z 456.484,A -85,B 0,C 180,E1 -16641.634,E2 -16641.634} C_VEL
LIN {X 0,Y 289.784,Z 458.492,A -85,B 0,C 180,E1 -16643.919,E2 -16643.919} C_VEL
LIN {X 0,Y 289.889,Z 459.303,A -85,B 0,C 180,E1 -16645.829,E2 -16645.829} C_VEL
LIN {X 0,Y 290.135,Z 459.422,A -85,B 0,C 180,E1 -16647.223,E2 -16647.223} C_VEL
LIN {X 0,Y 290.367,Z 459.086,A -85,B 0,C 180,E1 -16648.613,E2 -16648.613} C_VEL
LIN {X 0,Y 290.493,Z 457.254,A -85,B 0,C 180,E1 -16651.213,E2 -16651.213} C_VEL
LIN {X 0,Y 290.238,Z 457.879,A -85,B 0,C 180,E1 -16652.776,E2 -16652.776} C_VEL
LIN {X 0,Y 289.973,Z 457.781,A -85,B 0,C 180,E1 -16654.17,E2 -16654.17} C_VEL
LIN {X 0,Y 289.938,Z 457.028,A -85,B 0,C 180,E1 -16655.564,E2 -16655.564} C_VEL
LIN {X 0,Y 290.011,Z 454.612,A -85,B 0,C 180,E1 -16657.659,E2 -16657.659} C_VEL
LIN {X 0,Y 290.363,Z 450.688,A -85,B 0,C 180,E1 -16659.755,E2 -16659.755} C_VEL
LIN {X 0,Y 291.049,Z 445.057,A -85,B 0,C 180,E1 -16661.844,E2 -16661.844} C_VEL
LIN {X 0,Y 291.997,Z 438.715,A -85,B 0,C 180,E1 -16663.572,E2 -16663.572} C_VEL
LIN {X 0,Y 293.23,Z 430.634,A -85,B 0,C 180,E1 -16665.286,E2 -16665.286} C_VEL
LIN {X 0,Y 294.364,Z 422.383,A -85,B 0,C 180,E1 -16666.649,E2 -16666.649} C_VEL
LIN {X 0,Y 295.381,Z 413.627,A -85,B 0,C 180,E1 -16667.782,E2 -16667.782} C_VEL
LIN {X 0,Y 296.506,Z 403.815,A -85,B 0,C 180,E1 -16668.752,E2 -16668.752} C_VEL
LIN {X 0,Y 296.36,Z 394.426,A -85,B 0,C 180,E1 -16669.548,E2 -16669.548} C_VEL
LIN {X 0,Y 295.524,Z 387.151,A -85,B 0,C 180,E1 -16670.172,E2 -16670.172} C_VEL
LIN {X 0,Y 296.779,Z 377.748,A -85,B 0,C 180,E1 -16671.562,E2 -16671.562} C_VEL
LIN {X 0,Y 296.702,Z 368.308,A -85,B 0,C 180,E1 -16673.375,E2 -16673.375} C_VEL
LIN {X 0,Y 296.892,Z 359.783,A -85,B 0,C 180,E1 -16675.22,E2 -16675.22} C_VEL
LIN {X 0,Y 297.193,Z 353.701,A -85,B 0,C 180,E1 -16676.7,E2 -16676.7} C_VEL
LIN {X 0,Y 298.261,Z 343.118,A -85,B 0,C 180,E1 -16679.659,E2 -16679.659} C_VEL
LIN {X 0,Y 299.039,Z 338.103,A -85,B 0,C 180,E1 -16681.396,E2 -16681.396} C_VEL
LIN {X 0,Y 298.356,Z 332.742,A -85,B 0,C 180,E1 -16684.465,E2 -16684.465} C_VEL
LIN {X 0,Y 298.404,Z 329.578,A -85,B 0,C 180,E1 -16686.794,E2 -16686.794} C_VEL
LIN {X 0,Y 298.519,Z 327.444,A -85,B 0,C 180,E1 -16689.019,E2 -16689.019} C_VEL
LIN {X 0,Y 298.43,Z 326.56,A -85,B 0,C 180,E1 -16691.254,E2 -16691.254} C_VEL
LIN {X 0,Y 298.171,Z 326.334,A -85,B 0,C 180,E1 -16693.121,E2 -16693.121} C_VEL
LIN {X 0,Y 298.129,Z 326.601,A -85,B 0,C 180,E1 -16695.009,E2 -16695.009} C_VEL
LIN {X 0,Y 298.179,Z 328.258,A -85,B 0,C 180,E1 -16698.959,E2 -16698.959} C_VEL
LIN {X 0,Y 298.492,Z 330.639,A -85,B 0,C 180,E1 -16702.252,E2 -16702.252} C_VEL
LIN {X 0,Y 298.915,Z 334.056,A -85,B 0,C 180,E1 -16705.646,E2 -16705.646} C_VEL
LIN {X 0,Y 299.009,Z 336.481,A -85,B 0,C 180,E1 -16707.796,E2 -16707.796} C_VEL
LIN {X 0,Y 298.81,Z 338.965,A -85,B 0,C 180,E1 -16709.622,E2 -16709.622} C_VEL
LIN {X 0,Y 297.442,Z 345.65,A -85,B 0,C 180,E1 -16713.88,E2 -16713.88} C_VEL
LIN {X 0,Y 296.27,Z 353.155,A -85,B 0,C 180,E1 -16718.425,E2 -16718.425} C_VEL
LIN {X 0,Y 295.962,Z 355.997,A -85,B 0,C 180,E1 -16720.016,E2 -16720.016} C_VEL
LIN {X 0,Y 299.17,Z 364.946,A -85,B 0,C 180,E1 -16721.438,E2 -16721.438} C_VEL
LIN {X 0,Y 301.332,Z 374.012,A -85,B 0,C 180,E1 -16722.99,E2 -16722.99} C_VEL
LIN {X 0,Y 301.789,Z 377.352,A -85,B 0,C 180,E1 -16723.599,E2 -16723.599} C_VEL
LIN {X 0,Y 300.354,Z 384.941,A -85,B 0,C 180,E1 -16724.827,E2 -16724.827} C_VEL
LIN {X 0,Y 298.402,Z 392.347,A -85,B 0,C 180,E1 -16726.376,E2 -16726.376} C_VEL
LIN {X 0,Y 296.712,Z 398.172,A -85,B 0,C 180,E1 -16728.037,E2 -16728.037} C_VEL
LIN {X 0,Y 295.247,Z 402.584,A -85,B 0,C 180,E1 -16729.714,E2 -16729.714} C_VEL
LIN {X 0,Y 293.614,Z 406.098,A -85,B 0,C 180,E1 -16731.741,E2 -16731.741} C_VEL
LIN {X 0,Y 292.598,Z 407.572,A -85,B 0,C 180,E1 -16733.101,E2 -16733.101} C_VEL
LIN {X 0,Y 291.755,Z 408.347,A -85,B 0,C 180,E1 -16734.469,E2 -16734.469} C_VEL
LIN {X 0,Y 291.087,Z 408.439,A -85,B 0,C 180,E1 -16735.845,E2 -16735.845} C_VEL
LIN {X 0,Y 290.633,Z 407.845,A -85,B 0,C 180,E1 -16737.226,E2 -16737.226} C_VEL
LIN {X 0,Y 290.343,Z 406.562,A -85,B 0,C 180,E1 -16738.611,E2 -16738.611} C_VEL
LIN {X 0,Y 290.121,Z 403.284,A -85,B 0,C 180,E1 -16740.692,E2 -16740.692} C_VEL
LIN {X 0,Y 290.085,Z 400.186,A -85,B 0,C 180,E1 -16742.081,E2 -16742.081} C_VEL
LIN {X 0,Y 290.189,Z 395.005,A -85,B 0,C 180,E1 -16743.817,E2 -16743.817} C_VEL
LIN {X 0,Y 290.473,Z 389.748,A -85,B 0,C 180,E1 -16745.204,E2 -16745.204} C_VEL
LIN {X 0,Y 290.691,Z 383.093,A -85,B 0,C 180,E1 -16746.593,E2 -16746.593} C_VEL
LIN {X 0,Y 290.878,Z 375.447,A -85,B 0,C 180,E1 -16747.854,E2 -16747.854} C_VEL
LIN {X 0,Y 291.12,Z 366.245,A -85,B 0,C 180,E1 -16749.026,E2 -16749.026} C_VEL
LIN {X 0,Y 291.416,Z 356.263,A -85,B 0,C 180,E1 -16749.98,E2 -16749.98} C_VEL
LIN {X 0,Y 290.725,Z 348.713,A -85,B 0,C 180,E1 -16750.532,E2 -16750.532} C_VEL
LIN {X 0,Y 290.845,Z 339.521,A -85,B 0,C 180,E1 -16754.857,E2 -16754.857} C_VEL
LIN {X 0,Y 290.991,Z 329.582,A -85,B 0,C 180,E1 -16759.622,E2 -16759.622} C_VEL
LIN {X 0,Y 291.141,Z 321.672,A -85,B 0,C 180,E1 -16763.465,E2 -16763.465} C_VEL
LIN {X 0,Y 291.395,Z 313.903,A -85,B 0,C 180,E1 -16767.272,E2 -16767.272} C_VEL
LIN {X 0,Y 291.566,Z 308.164,A -85,B 0,C 180,E1 -16770.13,E2 -16770.13} C_VEL
LIN {X 0,Y 291.362,Z 308.19,A -85,B 0,C 180,E1 -16774.903,E2 -16774.903} C_VEL
LIN {X 0,Y 291.353,Z 308.195,A -85,B 0,C 180,E1 -16777.248,E2 -16777.248} C_VEL
LIN {X 0,Y 291.294,Z 308.199,A -85,B 0,C 180,E1 -16780.646,E2 -16780.646} C_VEL
LIN {X 0,Y 291.283,Z 308.199,A -85,B 0,C 180,E1 -16784.4,E2 -16784.4} C_VEL
LIN {X 0,Y 291.319,Z 308.196,A -85,B 0,C 180,E1 -16788.403,E2 -16788.403} C_VEL
LIN {X 0,Y 291.345,Z 308.193,A -85,B 0,C 180,E1 -16791.157,E2 -16791.157} C_VEL
LIN {X 0,Y 291.353,Z 308.194,A -85,B 0,C 180,E1 -16794.625,E2 -16794.625} C_VEL
LIN {X 0,Y 291.363,Z 308.189,A -85,B 0,C 180,E1 -16797.949,E2 -16797.949} C_VEL
LIN {X 0,Y 291.373,Z 308.188,A -85,B 0,C 180,E1 -16801.157,E2 -16801.157} C_VEL
LIN {X 0,Y 291.407,Z 308.186,A -85,B 0,C 180,E1 -16804.271,E2 -16804.271} C_VEL
LIN {X 0,Y 291.379,Z 308.186,A -85,B 0,C 180,E1 -16807.299,E2 -16807.299} C_VEL
LIN {X 0,Y 291.448,Z 308.181,A -85,B 0,C 180,E1 -16810.269,E2 -16810.269} C_VEL
LIN {X 0,Y 291.544,Z 308.169,A -85,B 0,C 180,E1 -16814.623,E2 -16814.623} C_VEL
LIN {X 0,Y 291.517,Z 308.17,A -85,B 0,C 180,E1 -16818.88,E2 -16818.88} C_VEL
LIN {X 0,Y 291.64,Z 308.156,A -85,B 0,C 180,E1 -16821.686,E2 -16821.686} C_VEL
LIN {X 0,Y 291.588,Z 308.162,A -85,B 0,C 180,E1 -16824.468,E2 -16824.468} C_VEL
LIN {X 0,Y 291.858,Z 308.128,A -85,B 0,C 180,E1 -16828.62,E2 -16828.62} C_VEL
LIN {X 0,Y 291.858,Z 308.128,A -85,B 0,C 180,E1 -16831.38,E2 -16831.38} C_VEL
LIN {X 0,Y 291.676,Z 308.15,A -85,B 0,C 180,E1 -16836.92,E2 -16836.92} C_VEL
LIN {X 0,Y 291.556,Z 308.169,A -85,B 0,C 180,E1 -16839.714,E2 -16839.714} C_VEL
LIN {X 0,Y 291.51,Z 308.173,A -85,B 0,C 180,E1 -16843.951,E2 -16843.951} C_VEL
LIN {X 0,Y 291.476,Z 308.175,A -85,B 0,C 180,E1 -16846.819,E2 -16846.819} C_VEL
LIN {X 0,Y 291.44,Z 308.181,A -85,B 0,C 180,E1 -16849.876,E2 -16849.876} C_VEL
LIN {X 0,Y 291.39,Z 308.186,A -85,B 0,C 180,E1 -16854.206,E2 -16854.206} C_VEL
LIN {X 0,Y 291.413,Z 308.187,A -85,B 0,C 180,E1 -16857.273,E2 -16857.273} C_VEL
LIN {X 0,Y 291.328,Z 308.192,A -85,B 0,C 180,E1 -16860.438,E2 -16860.438} C_VEL
LIN {X 0,Y 291.336,Z 308.194,A -85,B 0,C 180,E1 -16863.7,E2 -16863.7} C_VEL
LIN {X 0,Y 291.369,Z 308.192,A -85,B 0,C 180,E1 -16867.256,E2 -16867.256} C_VEL
LIN {X 0,Y 291.325,Z 308.195,A -85,B 0,C 180,E1 -16870.644,E2 -16870.644} C_VEL
LIN {X 0,Y 291.282,Z 308.2,A -85,B 0,C 180,E1 -16874.404,E2 -16874.404} C_VEL
LIN {X 0,Y 291.288,Z 308.199,A -85,B 0,C 180,E1 -16878.413,E2 -16878.413} C_VEL
LIN {X 0,Y 291.328,Z 308.196,A -85,B 0,C 180,E1 -16881.157,E2 -16881.157} C_VEL
LIN {X 0,Y 291.35,Z 308.194,A -85,B 0,C 180,E1 -16884.627,E2 -16884.627} C_VEL
LIN {X 0,Y 291.576,Z 308.18,A -85,B 0,C 180,E1 -16888.182,E2 -16888.182} C_VEL
LIN {X 0,Y 291.703,Z 311.028,A -85,B 0,C 180,E1 -16890.152,E2 -16890.152} C_VEL
LIN {X 0,Y 291.326,Z 315.566,A -85,B 0,C 180,E1 -16893.202,E2 -16893.202} C_VEL
LIN {X 0,Y 290.965,Z 320.739,A -85,B 0,C 180,E1 -16896.615,E2 -16896.615} C_VEL
LIN {X 0,Y 290.625,Z 326.872,A -85,B 0,C 180,E1 -16900.581,E2 -16900.581} C_VEL
LIN {X 0,Y 290.309,Z 333.151,A -85,B 0,C 180,E1 -16904.558,E2 -16904.558} C_VEL
LIN {X 0,Y 290.2,Z 337.999,A -85,B 0,C 180,E1 -16907.502,E2 -16907.502} C_VEL
LIN {X 0,Y 291.312,Z 349.949,A -85,B 0,C 180,E1 -16908.433,E2 -16908.433} C_VEL
LIN {X 0,Y 292.008,Z 356.469,A -85,B 0,C 180,E1 -16909.076,E2 -16909.076} C_VEL
LIN {X 0,Y 291.554,Z 366.624,A -85,B 0,C 180,E1 -16910.288,E2 -16910.288} C_VEL
LIN {X 0,Y 291.132,Z 375.846,A -85,B 0,C 180,E1 -16911.674,E2 -16911.674} C_VEL
LIN {X 0,Y 290.81,Z 383.331,A -85,B 0,C 180,E1 -16913.062,E2 -16913.062} C_VEL
LIN {X 0,Y 290.494,Z 390.863,A -85,B 0,C 180,E1 -16914.797,E2 -16914.797} C_VEL
LIN {X 0,Y 290.169,Z 396.786,A -85,B 0,C 180,E1 -16916.53,E2 -16916.53} C_VEL
LIN {X 0,Y 290.097,Z 402.145,A -85,B 0,C 180,E1 -16918.614,E2 -16918.614} C_VEL
LIN {X 0,Y 290.253,Z 405.894,A -85,B 0,C 180,E1 -16920.695,E2 -16920.695} C_VEL
LIN {X 0,Y 290.667,Z 408.189,A -85,B 0,C 180,E1 -16922.774,E2 -16922.774} C_VEL
LIN {X 0,Y 291.183,Z 408.966,A -85,B 0,C 180,E1 -16924.336,E2 -16924.336} C_VEL
LIN {X 0,Y 290.864,Z 409.18,A -85,B 0,C 180,E1 -16925.123,E2 -16925.123} C_VEL
LIN {X 0,Y 288.692,Z 409.464,A -85,B 0,C 180,E1 -16926.396,E2 -16926.396} C_VEL
LIN {X 0,Y 286.693,Z 409.325,A -85,B 0,C 180,E1 -16927.679,E2 -16927.679} C_VEL
LIN {X 0,Y 286.634,Z 408.743,A -85,B 0,C 180,E1 -16928.464,E2 -16928.464} C_VEL
LIN {X 0,Y 288.551,Z 406.259,A -85,B 0,C 180,E1 -16930.527,E2 -16930.527} C_VEL
LIN {X 0,Y 290.657,Z 402.376,A -85,B 0,C 180,E1 -16932.571,E2 -16932.571} C_VEL
LIN {X 0,Y 293.101,Z 396.954,A -85,B 0,C 180,E1 -16934.584,E2 -16934.584} C_VEL
LIN {X 0,Y 296.001,Z 389.788,A -85,B 0,C 180,E1 -16936.556,E2 -16936.556} C_VEL
LIN {X 0,Y 298.066,Z 383.832,A -85,B 0,C 180,E1 -16937.851,E2 -16937.851} C_VEL
LIN {X 0,Y 298.229,Z 378.861,A -85,B 0,C 180,E1 -16939.049,E2 -16939.049} C_VEL
LIN {X 0,Y 297.489,Z 371.805,A -85,B 0,C 180,E1 -16940.756,E2 -16940.756} C_VEL
LIN {X 0,Y 295.748,Z 363.791,A -85,B 0,C 180,E1 -16942.718,E2 -16942.718} C_VEL
LIN {X 0,Y 292.635,Z 354.41,A -85,B 0,C 180,E1 -16945.148,E2 -16945.148} C_VEL
LIN {X 0,Y 291.034,Z 350.69,A -85,B 0,C 180,E1 -16946.19,E2 -16946.19} C_VEL
LIN {X 0,Y 289.77,Z 347.128,A -85,B 0,C 180,E1 -16947.198,E2 -16947.198} C_VEL
LIN {X 0,Y 290.554,Z 345.539,A -85,B 0,C 180,E1 -16949.45,E2 -16949.45} C_VEL
LIN {X 0,Y 291.456,Z 343.876,A -85,B 0,C 180,E1 -16952.438,E2 -16952.438} C_VEL
LIN {X 0,Y 291.887,Z 342.873,A -85,B 0,C 180,E1 -16955.302,E2 -16955.302} C_VEL
LIN {X 0,Y 292.222,Z 342.454,A -85,B 0,C 180,E1 -16958.706,E2 -16958.706} C_VEL
LIN {X 0,Y 292.594,Z 342.862,A -85,B 0,C 180,E1 -16962.266,E2 -16962.266} C_VEL
LIN {X 0,Y 293.137,Z 344.317,A -85,B 0,C 180,E1 -16965.995,E2 -16965.995} C_VEL
LIN {X 0,Y 293.473,Z 345.487,A -85,B 0,C 180,E1 -16967.936,E2 -16967.936} C_VEL
LIN {X 0,Y 294.155,Z 348.552,A -85,B 0,C 180,E1 -16971.596,E2 -16971.596} C_VEL
LIN {X 0,Y 294.968,Z 352.522,A -85,B 0,C 180,E1 -16975.122,E2 -16975.122} C_VEL
LIN {X 0,Y 295.285,Z 354.835,A -85,B 0,C 180,E1 -16976.81,E2 -16976.81} C_VEL
LIN {X 0,Y 294.363,Z 357.532,A -85,B 0,C 180,E1 -16978.314,E2 -16978.314} C_VEL
LIN {X 0,Y 294.001,Z 358.697,A -85,B 0,C 180,E1 -16978.797,E2 -16978.797} C_VEL
LIN {X 0,Y 296.835,Z 372.149,A -85,B 0,C 180,E1 -16980.839,E2 -16980.839} C_VEL
LIN {X 0,Y 298.335,Z 384.449,A -85,B 0,C 180,E1 -16982.644,E2 -16982.644} C_VEL
LIN {X 0,Y 298.439,Z 396,A -85,B 0,C 180,E1 -16984.317,E2 -16984.317} C_VEL
LIN {X 0,Y 297.466,Z 404.53,A -85,B 0,C 180,E1 -16985.578,E2 -16985.578} C_VEL
LIN {X 0,Y 295.48,Z 412.964,A -85,B 0,C 180,E1 -16986.893,E2 -16986.893} C_VEL
LIN {X 0,Y 292.11,Z 423.671,A -85,B 0,C 180,E1 -16988.845,E2 -16988.845} C_VEL
LIN {X 0,Y 289.325,Z 432.286,A -85,B 0,C 180,E1 -16990.857,E2 -16990.857} C_VEL
LIN {X 0,Y 286.742,Z 440.405,A -85,B 0,C 180,E1 -16993.262,E2 -16993.262} C_VEL
LIN {X 0,Y 284.908,Z 446.785,A -85,B 0,C 180,E1 -16995.719,E2 -16995.719} C_VEL
LIN {X 0,Y 283.648,Z 451.076,A -85,B 0,C 180,E1 -16997.842,E2 -16997.842} C_VEL
LIN {X 0,Y 282.988,Z 454.354,A -85,B 0,C 180,E1 -16999.989,E2 -16999.989} C_VEL
LIN {X 0,Y 282.769,Z 456.007,A -85,B 0,C 180,E1 -17001.424,E2 -17001.424} C_VEL
LIN {X 0,Y 282.738,Z 458.105,A -85,B 0,C 180,E1 -17004.294,E2 -17004.294} C_VEL
LIN {X 0,Y 282.815,Z 458.531,A -85,B 0,C 180,E1 -17005.725,E2 -17005.725} C_VEL
LIN {X 0,Y 283.07,Z 458.536,A -85,B 0,C 180,E1 -17007.154,E2 -17007.154} C_VEL
LIN {X 0,Y 283.32,Z 458.133,A -85,B 0,C 180,E1 -17008.579,E2 -17008.579} C_VEL
LIN {X 0,Y 283.467,Z 456.283,A -85,B 0,C 180,E1 -17011.065,E2 -17011.065} C_VEL
LIN {X 0,Y 283.429,Z 456.208,A -85,B 0,C 180,E1 -17011.421,E2 -17011.421} C_VEL
LIN {X 0,Y 283.182,Z 456.965,A -85,B 0,C 180,E1 -17012.845,E2 -17012.845} C_VEL
LIN {X 0,Y 282.897,Z 457.032,A -85,B 0,C 180,E1 -17014.274,E2 -17014.274} C_VEL
LIN {X 0,Y 282.88,Z 455.912,A -85,B 0,C 180,E1 -17016.384,E2 -17016.384} C_VEL
LIN {X 0,Y 283.024,Z 453.304,A -85,B 0,C 180,E1 -17018.569,E2 -17018.569} C_VEL
LIN {X 0,Y 283.34,Z 450.709,A -85,B 0,C 180,E1 -17019.999,E2 -17019.999} C_VEL
LIN {X 0,Y 283.932,Z 446.384,A -85,B 0,C 180,E1 -17021.783,E2 -17021.783} C_VEL
LIN {X 0,Y 284.913,Z 440.83,A -85,B 0,C 180,E1 -17023.553,E2 -17023.553} C_VEL
LIN {X 0,Y 286.206,Z 433.566,A -85,B 0,C 180,E1 -17025.306,E2 -17025.306} C_VEL
LIN {X 0,Y 287.538,Z 425.397,A -85,B 0,C 180,E1 -17026.873,E2 -17026.873} C_VEL
LIN {X 0,Y 289.021,Z 415.76,A -85,B 0,C 180,E1 -17028.279,E2 -17028.279} C_VEL
LIN {X 0,Y 290.246,Z 406.785,A -85,B 0,C 180,E1 -17029.263,E2 -17029.263} C_VEL
LIN {X 0,Y 290.665,Z 399.43,A -85,B 0,C 180,E1 -17029.97,E2 -17029.97} C_VEL
LIN {X 0,Y 289.797,Z 388.333,A -85,B 0,C 180,E1 -17030.983,E2 -17030.983} C_VEL
LIN {X 0,Y 289.688,Z 386.301,A -85,B 0,C 180,E1 -17031.154,E2 -17031.154} C_VEL
LIN {X 0,Y 290.691,Z 379.078,A -85,B 0,C 180,E1 -17032.303,E2 -17032.303} C_VEL
LIN {X 0,Y 290.951,Z 367.639,A -85,B 0,C 180,E1 -17034.625,E2 -17034.625} C_VEL
LIN {X 0,Y 291.421,Z 358.356,A -85,B 0,C 180,E1 -17036.833,E2 -17036.833} C_VEL
LIN {X 0,Y 292.507,Z 347.754,A -85,B 0,C 180,E1 -17039.835,E2 -17039.835} C_VEL
LIN {X 0,Y 293.498,Z 342.103,A -85,B 0,C 180,E1 -17041.79,E2 -17041.79} C_VEL
LIN {X 0,Y 292.842,Z 336.035,A -85,B 0,C 180,E1 -17045.314,E2 -17045.314} C_VEL
LIN {X 0,Y 292.889,Z 333.176,A -85,B 0,C 180,E1 -17047.639,E2 -17047.639} C_VEL
LIN {X 0,Y 292.953,Z 331.453,A -85,B 0,C 180,E1 -17049.852,E2 -17049.852} C_VEL
LIN {X 0,Y 292.579,Z 330.645,A -85,B 0,C 180,E1 -17052.267,E2 -17052.267} C_VEL
LIN {X 0,Y 292.394,Z 330.689,A -85,B 0,C 180,E1 -17054.191,E2 -17054.191} C_VEL
LIN {X 0,Y 292.22,Z 331.58,A -85,B 0,C 180,E1 -17057.667,E2 -17057.667} C_VEL
LIN {X 0,Y 292.342,Z 333.645,A -85,B 0,C 180,E1 -17061.312,E2 -17061.312} C_VEL
LIN {X 0,Y 292.502,Z 335.019,A -85,B 0,C 180,E1 -17063.08,E2 -17063.08} C_VEL
LIN {X 0,Y 292.702,Z 338.393,A -85,B 0,C 180,E1 -17066.477,E2 -17066.477} C_VEL
LIN {X 0,Y 292.564,Z 341.281,A -85,B 0,C 180,E1 -17068.902,E2 -17068.902} C_VEL
LIN {X 0,Y 291.53,Z 345.766,A -85,B 0,C 180,E1 -17071.958,E2 -17071.958} C_VEL
LIN {X 0,Y 290.201,Z 352.812,A -85,B 0,C 180,E1 -17076.446,E2 -17076.446} C_VEL
LIN {X 0,Y 289.647,Z 357.088,A -85,B 0,C 180,E1 -17078.962,E2 -17078.962} C_VEL
LIN {X 0,Y 292.938,Z 366.289,A -85,B 0,C 180,E1 -17080.558,E2 -17080.558} C_VEL
LIN {X 0,Y 294.796,Z 373.913,A -85,B 0,C 180,E1 -17081.944,E2 -17081.944} C_VEL
LIN {X 0,Y 295.594,Z 380.161,A -85,B 0,C 180,E1 -17083.148,E2 -17083.148} C_VEL
LIN {X 0,Y 293.938,Z 387.365,A -85,B 0,C 180,E1 -17084.409,E2 -17084.409} C_VEL
LIN {X 0,Y 292.188,Z 393.432,A -85,B 0,C 180,E1 -17085.725,E2 -17085.725} C_VEL
LIN {X 0,Y 290.352,Z 399.175,A -85,B 0,C 180,E1 -17087.416,E2 -17087.416} C_VEL
LIN {X 0,Y 289.05,Z 402.717,A -85,B 0,C 180,E1 -17088.782,E2 -17088.782} C_VEL
LIN {X 0,Y 287.823,Z 405.443,A -85,B 0,C 180,E1 -17090.157,E2 -17090.157} C_VEL
LIN {X 0,Y 286.73,Z 407.423,A -85,B 0,C 180,E1 -17091.541,E2 -17091.541} C_VEL
LIN {X 0,Y 285.637,Z 408.697,A -85,B 0,C 180,E1 -17092.932,E2 -17092.932} C_VEL
LIN {X 0,Y 284.749,Z 409.268,A -85,B 0,C 180,E1 -17094.332,E2 -17094.332} C_VEL
LIN {X 0,Y 284.07,Z 409.153,A -85,B 0,C 180,E1 -17095.742,E2 -17095.742} C_VEL
LIN {X 0,Y 283.575,Z 408.362,A -85,B 0,C 180,E1 -17097.157,E2 -17097.157} C_VEL
LIN {X 0,Y 283.162,Z 405.937,A -85,B 0,C 180,E1 -17099.287,E2 -17099.287} C_VEL
LIN {X 0,Y 283.034,Z 403.407,A -85,B 0,C 180,E1 -17100.71,E2 -17100.71} C_VEL
LIN {X 0,Y 282.998,Z 398.043,A -85,B 0,C 180,E1 -17102.845,E2 -17102.845} C_VEL
LIN {X 0,Y 283.262,Z 391.929,A -85,B 0,C 180,E1 -17104.623,E2 -17104.623} C_VEL
LIN {X 0,Y 283.553,Z 385.717,A -85,B 0,C 180,E1 -17106.045,E2 -17106.045} C_VEL
LIN {X 0,Y 283.72,Z 377.105,A -85,B 0,C 180,E1 -17107.571,E2 -17107.571} C_VEL
LIN {X 0,Y 283.99,Z 368.845,A -85,B 0,C 180,E1 -17108.716,E2 -17108.716} C_VEL
LIN {X 0,Y 284.235,Z 358.6,A -85,B 0,C 180,E1 -17109.785,E2 -17109.785} C_VEL
LIN {X 0,Y 284.217,Z 354.074,A -85,B 0,C 180,E1 -17110.146,E2 -17110.146} C_VEL
LIN {X 0,Y 283.672,Z 349.343,A -85,B 0,C 180,E1 -17110.481,E2 -17110.481} C_VEL
LIN {X 0,Y 283.74,Z 341.222,A -85,B 0,C 180,E1 -17114.339,E2 -17114.339} C_VEL
LIN {X 0,Y 283.863,Z 332.033,A -85,B 0,C 180,E1 -17118.773,E2 -17118.773} C_VEL
LIN {X 0,Y 284.03,Z 324.314,A -85,B 0,C 180,E1 -17122.55,E2 -17122.55} C_VEL
LIN {X 0,Y 284.314,Z 316.463,A -85,B 0,C 180,E1 -17126.417,E2 -17126.417} C_VEL
LIN {X 0,Y 284.53,Z 309.04,A -85,B 0,C 180,E1 -17130.172,E2 -17130.172} C_VEL
LIN {X 0,Y 284.331,Z 309.068,A -85,B 0,C 180,E1 -17135.345,E2 -17135.345} C_VEL
LIN {X 0,Y 284.292,Z 309.07,A -85,B 0,C 180,E1 -17138.169,E2 -17138.169} C_VEL
LIN {X 0,Y 284.231,Z 309.076,A -85,B 0,C 180,E1 -17142.115,E2 -17142.115} C_VEL
LIN {X 0,Y 284.247,Z 309.075,A -85,B 0,C 180,E1 -17146.187,E2 -17146.187} C_VEL
LIN {X 0,Y 284.299,Z 309.068,A -85,B 0,C 180,E1 -17150.022,E2 -17150.022} C_VEL
LIN {X 0,Y 284.324,Z 309.066,A -85,B 0,C 180,E1 -17153.613,E2 -17153.613} C_VEL
LIN {X 0,Y 284.299,Z 309.07,A -85,B 0,C 180,E1 -17157.188,E2 -17157.188} C_VEL
LIN {X 0,Y 284.349,Z 309.064,A -85,B 0,C 180,E1 -17160.375,E2 -17160.375} C_VEL
LIN {X 0,Y 284.368,Z 309.06,A -85,B 0,C 180,E1 -17163.586,E2 -17163.586} C_VEL
LIN {X 0,Y 284.359,Z 309.064,A -85,B 0,C 180,E1 -17166.706,E2 -17166.706} C_VEL
LIN {X 0,Y 284.393,Z 309.057,A -85,B 0,C 180,E1 -17171.261,E2 -17171.261} C_VEL
LIN {X 0,Y 284.482,Z 309.05,A -85,B 0,C 180,E1 -17174.458,E2 -17174.458} C_VEL
LIN {X 0,Y 284.471,Z 309.049,A -85,B 0,C 180,E1 -17178.601,E2 -17178.601} C_VEL
LIN {X 0,Y 284.597,Z 309.032,A -85,B 0,C 180,E1 -17181.479,E2 -17181.479} C_VEL
LIN {X 0,Y 284.558,Z 309.039,A -85,B 0,C 180,E1 -17184.33,E2 -17184.33} C_VEL
LIN {X 0,Y 284.825,Z 309.004,A -85,B 0,C 180,E1 -17188.586,E2 -17188.586} C_VEL
LIN {X 0,Y 284.826,Z 309.004,A -85,B 0,C 180,E1 -17191.414,E2 -17191.414} C_VEL
LIN {X 0,Y 284.631,Z 309.028,A -85,B 0,C 180,E1 -17197.092,E2 -17197.092} C_VEL
LIN {X 0,Y 284.502,Z 309.047,A -85,B 0,C 180,E1 -17199.958,E2 -17199.958} C_VEL
LIN {X 0,Y 284.47,Z 309.048,A -85,B 0,C 180,E1 -17204.303,E2 -17204.303} C_VEL
LIN {X 0,Y 284.415,Z 309.056,A -85,B 0,C 180,E1 -17207.249,E2 -17207.249} C_VEL
LIN {X 0,Y 284.37,Z 309.06,A -85,B 0,C 180,E1 -17210.243,E2 -17210.243} C_VEL
LIN {X 0,Y 284.359,Z 309.063,A -85,B 0,C 180,E1 -17213.876,E2 -17213.876} C_VEL
LIN {X 0,Y 284.388,Z 309.061,A -85,B 0,C 180,E1 -17217.175,E2 -17217.175} C_VEL
LIN {X 0,Y 284.287,Z 309.074,A -85,B 0,C 180,E1 -17221.276,E2 -17221.276} C_VEL
LIN {X 0,Y 284.333,Z 309.068,A -85,B 0,C 180,E1 -17225.35,E2 -17225.35} C_VEL
LIN {X 0,Y 284.304,Z 309.067,A -85,B 0,C 180,E1 -17228.17,E2 -17228.17} C_VEL
LIN {X 0,Y 284.261,Z 309.074,A -85,B 0,C 180,E1 -17232.126,E2 -17232.126} C_VEL
LIN {X 0,Y 284.248,Z 309.075,A -85,B 0,C 180,E1 -17236.191,E2 -17236.191} C_VEL
LIN {X 0,Y 284.277,Z 309.072,A -85,B 0,C 180,E1 -17240.032,E2 -17240.032} C_VEL
LIN {X 0,Y 284.315,Z 309.067,A -85,B 0,C 180,E1 -17243.614,E2 -17243.614} C_VEL
LIN {X 0,Y 284.534,Z 309.045,A -85,B 0,C 180,E1 -17248.135,E2 -17248.135} C_VEL
LIN {X 0,Y 284.63,Z 312.287,A -85,B 0,C 180,E1 -17250.41,E2 -17250.41} C_VEL
LIN {X 0,Y 284.133,Z 318.083,A -85,B 0,C 180,E1 -17254.353,E2 -17254.353} C_VEL
LIN {X 0,Y 283.754,Z 323.845,A -85,B 0,C 180,E1 -17258.193,E2 -17258.193} C_VEL
LIN {X 0,Y 283.426,Z 329.586,A -85,B 0,C 180,E1 -17261.946,E2 -17261.946} C_VEL
LIN {X 0,Y 283.125,Z 336.501,A -85,B 0,C 180,E1 -17266.362,E2 -17266.362} C_VEL
LIN {X 0,Y 283.121,Z 338.163,A -85,B 0,C 180,E1 -17267.412,E2 -17267.412} C_VEL
LIN {X 0,Y 284.209,Z 350.491,A -85,B 0,C 180,E1 -17268.411,E2 -17268.411} C_VEL
LIN {X 0,Y 284.862,Z 357.79,A -85,B 0,C 180,E1 -17269.159,E2 -17269.159} C_VEL
LIN {X 0,Y 284.375,Z 367.772,A -85,B 0,C 180,E1 -17270.399,E2 -17270.399} C_VEL
LIN {X 0,Y 283.982,Z 376.5,A -85,B 0,C 180,E1 -17271.751,E2 -17271.751} C_VEL
LIN {X 0,Y 283.698,Z 384.335,A -85,B 0,C 180,E1 -17273.244,E2 -17273.244} C_VEL
LIN {X 0,Y 283.361,Z 391.746,A -85,B 0,C 180,E1 -17275.022,E2 -17275.022} C_VEL
LIN {X 0,Y 283.01,Z 398.609,A -85,B 0,C 180,E1 -17277.155,E2 -17277.155} C_VEL
LIN {X 0,Y 283.057,Z 403.69,A -85,B 0,C 180,E1 -17279.291,E2 -17279.291} C_VEL
LIN {X 0,Y 283.292,Z 407.211,A -85,B 0,C 180,E1 -17281.423,E2 -17281.423} C_VEL
LIN {X 0,Y 283.606,Z 408.741,A -85,B 0,C 180,E1 -17282.843,E2 -17282.843} C_VEL
LIN {X 0,Y 284.167,Z 409.685,A -85,B 0,C 180,E1 -17284.446,E2 -17284.446} C_VEL
LIN {X 0,Y 284.742,Z 409.943,A -85,B 0,C 180,E1 -17285.668,E2 -17285.668} C_VEL
LIN {X 0,Y 285.611,Z 409.643,A -85,B 0,C 180,E1 -17287.069,E2 -17287.069} C_VEL
LIN {X 0,Y 286.634,Z 408.743,A -85,B 0,C 180,E1 -17288.464,E2 -17288.464} C_VEL
LIN {X 0,Y 286.995,Z 407.691,A -85,B 0,C 180,E1 -17289.621,E2 -17289.621} C_VEL
LIN {X 0,Y 286.026,Z 405.572,A -85,B 0,C 180,E1 -17291.557,E2 -17291.557} C_VEL
LIN {X 0,Y 285.287,Z 402.746,A -85,B 0,C 180,E1 -17293.452,E2 -17293.452} C_VEL
LIN {X 0,Y 285.976,Z 400.329,A -85,B 0,C 180,E1 -17294.519,E2 -17294.519} C_VEL
LIN {X 0,Y 288.51,Z 394.934,A -85,B 0,C 180,E1 -17296.27,E2 -17296.27} C_VEL
LIN {X 0,Y 291.73,Z 386.933,A -85,B 0,C 180,E1 -17298.253,E2 -17298.253} C_VEL
LIN {X 0,Y 292.314,Z 383.922,A -85,B 0,C 180,E1 -17298.988,E2 -17298.988} C_VEL
LIN {X 0,Y 291.889,Z 375.613,A -85,B 0,C 180,E1 -17301.173,E2 -17301.173} C_VEL
LIN {X 0,Y 290.561,Z 367.934,A -85,B 0,C 180,E1 -17303.2,E2 -17303.2} C_VEL
LIN {X 0,Y 288.183,Z 359.578,A -85,B 0,C 180,E1 -17305.534,E2 -17305.534} C_VEL
LIN {X 0,Y 285.666,Z 352.568,A -85,B 0,C 180,E1 -17307.665,E2 -17307.665} C_VEL
LIN {X 0,Y 284.062,Z 349.312,A -85,B 0,C 180,E1 -17308.847,E2 -17308.847} C_VEL
LIN {X 0,Y 283.787,Z 348.023,A -85,B 0,C 180,E1 -17309.233,E2 -17309.233} C_VEL
LIN {X 0,Y 284.406,Z 346.862,A -85,B 0,C 180,E1 -17311.263,E2 -17311.263} C_VEL
LIN {X 0,Y 284.854,Z 346.065,A -85,B 0,C 180,E1 -17312.98,E2 -17312.98} C_VEL
LIN {X 0,Y 285.324,Z 345.22,A -85,B 0,C 180,E1 -17316.241,E2 -17316.241} C_VEL
LIN {X 0,Y 285.75,Z 345.036,A -85,B 0,C 180,E1 -17319.754,E2 -17319.754} C_VEL
LIN {X 0,Y 286.117,Z 345.854,A -85,B 0,C 180,E1 -17323.456,E2 -17323.456} C_VEL
LIN {X 0,Y 286.746,Z 347.719,A -85,B 0,C 180,E1 -17327.333,E2 -17327.333} C_VEL
LIN {X 0,Y 287.309,Z 350.099,A -85,B 0,C 180,E1 -17330.506,E2 -17330.506} C_VEL
LIN {X 0,Y 288.078,Z 353.858,A -85,B 0,C 180,E1 -17334.161,E2 -17334.161} C_VEL
LIN {X 0,Y 288.511,Z 357.235,A -85,B 0,C 180,E1 -17336.764,E2 -17336.764} C_VEL
LIN {X 0,Y 288.402,Z 358.003,A -85,B 0,C 180,E1 -17337.14,E2 -17337.14} C_VEL
LIN {X 0,Y 290.594,Z 367.74,A -85,B 0,C 180,E1 -17338.851,E2 -17338.851} C_VEL
LIN {X 0,Y 292.4,Z 380.586,A -85,B 0,C 180,E1 -17340.923,E2 -17340.923} C_VEL
LIN {X 0,Y 292.851,Z 389.711,A -85,B 0,C 180,E1 -17342.35,E2 -17342.35} C_VEL
LIN {X 0,Y 292.435,Z 399.191,A -85,B 0,C 180,E1 -17343.833,E2 -17343.833} C_VEL
LIN {X 0,Y 291.019,Z 407.732,A -85,B 0,C 180,E1 -17345.191,E2 -17345.191} C_VEL
LIN {X 0,Y 287.895,Z 418.244,A -85,B 0,C 180,E1 -17347.009,E2 -17347.009} C_VEL
LIN {X 0,Y 285.072,Z 426.263,A -85,B 0,C 180,E1 -17348.676,E2 -17348.676} C_VEL
LIN {X 0,Y 282.234,Z 434.21,A -85,B 0,C 180,E1 -17350.735,E2 -17350.735} C_VEL
LIN {X 0,Y 279.609,Z 441.719,A -85,B 0,C 180,E1 -17353.199,E2 -17353.199} C_VEL
LIN {X 0,Y 277.515,Z 448.302,A -85,B 0,C 180,E1 -17356.079,E2 -17356.079} C_VEL
LIN {X 0,Y 276.331,Z 452.031,A -85,B 0,C 180,E1 -17358.26,E2 -17358.26} C_VEL
LIN {X 0,Y 275.697,Z 455.507,A -85,B 0,C 180,E1 -17361.202,E2 -17361.202} C_VEL
LIN {X 0,Y 275.655,Z 457.317,A -85,B 0,C 180,E1 -17363.907,E2 -17363.907} C_VEL
LIN {X 0,Y 275.745,Z 457.709,A -85,B 0,C 180,E1 -17365.615,E2 -17365.615} C_VEL
LIN {X 0,Y 276.005,Z 457.642,A -85,B 0,C 180,E1 -17367.081,E2 -17367.081} C_VEL
LIN {X 0,Y 276.28,Z 457.128,A -85,B 0,C 180,E1 -17368.542,E2 -17368.542} C_VEL
LIN {X 0,Y 276.485,Z 454.943,A -85,B 0,C 180,E1 -17371.274,E2 -17371.274} C_VEL
LIN {X 0,Y 276.144,Z 455.993,A -85,B 0,C 180,E1 -17372.918,E2 -17372.918} C_VEL
LIN {X 0,Y 275.83,Z 456.213,A -85,B 0,C 180,E1 -17374.384,E2 -17374.384} C_VEL
LIN {X 0,Y 275.791,Z 455.547,A -85,B 0,C 180,E1 -17376.351,E2 -17376.351} C_VEL
LIN {X 0,Y 275.977,Z 453.012,A -85,B 0,C 180,E1 -17378.789,E2 -17378.789} C_VEL
LIN {X 0,Y 276.535,Z 449.213,A -85,B 0,C 180,E1 -17380.988,E2 -17380.988} C_VEL
LIN {X 0,Y 277.615,Z 443.71,A -85,B 0,C 180,E1 -17383.17,E2 -17383.17} C_VEL
LIN {X 0,Y 278.885,Z 437.614,A -85,B 0,C 180,E1 -17384.97,E2 -17384.97} C_VEL
LIN {X 0,Y 280.12,Z 431.559,A -85,B 0,C 180,E1 -17386.395,E2 -17386.395} C_VEL
LIN {X 0,Y 281.617,Z 423.694,A -85,B 0,C 180,E1 -17387.871,E2 -17387.871} C_VEL
LIN {X 0,Y 282.921,Z 415.936,A -85,B 0,C 180,E1 -17389.047,E2 -17389.047} C_VEL
LIN {X 0,Y 284.573,Z 405.586,A -85,B 0,C 180,E1 -17390.228,E2 -17390.228} C_VEL
LIN {X 0,Y 284.763,Z 396.653,A -85,B 0,C 180,E1 -17391.159,E2 -17391.159} C_VEL
LIN {X 0,Y 284.061,Z 385.446,A -85,B 0,C 180,E1 -17392.205,E2 -17392.205} C_VEL
LIN {X 0,Y 284.642,Z 381.667,A -85,B 0,C 180,E1 -17392.838,E2 -17392.838} C_VEL
LIN {X 0,Y 285.086,Z 370.545,A -85,B 0,C 180,E1 -17395.167,E2 -17395.167} C_VEL
LIN {X 0,Y 285.755,Z 360.378,A -85,B 0,C 180,E1 -17397.696,E2 -17397.696} C_VEL
LIN {X 0,Y 286.946,Z 351.27,A -85,B 0,C 180,E1 -17400.363,E2 -17400.363} C_VEL
LIN {X 0,Y 287.691,Z 347.371,A -85,B 0,C 180,E1 -17401.683,E2 -17401.683} C_VEL
LIN {X 0,Y 287.825,Z 345.411,A -85,B 0,C 180,E1 -17402.493,E2 -17402.493} C_VEL
LIN {X 0,Y 287.346,Z 339.842,A -85,B 0,C 180,E1 -17405.945,E2 -17405.945} C_VEL
LIN {X 0,Y 287.396,Z 336.896,A -85,B 0,C 180,E1 -17408.505,E2 -17408.505} C_VEL
LIN {X 0,Y 287.196,Z 335.455,A -85,B 0,C 180,E1 -17410.657,E2 -17410.657} C_VEL
LIN {X 0,Y 286.767,Z 334.887,A -85,B 0,C 180,E1 -17413.332,E2 -17413.332} C_VEL
LIN {X 0,Y 286.415,Z 335.251,A -85,B 0,C 180,E1 -17416.6,E2 -17416.6} C_VEL
LIN {X 0,Y 286.329,Z 336.852,A -85,B 0,C 180,E1 -17420.342,E2 -17420.342} C_VEL
LIN {X 0,Y 286.42,Z 339.475,A -85,B 0,C 180,E1 -17423.919,E2 -17423.919} C_VEL
LIN {X 0,Y 286.462,Z 342.815,A -85,B 0,C 180,E1 -17427.332,E2 -17427.332} C_VEL
LIN {X 0,Y 286.13,Z 345.195,A -85,B 0,C 180,E1 -17429.281,E2 -17429.281} C_VEL
LIN {X 0,Y 284.514,Z 351.48,A -85,B 0,C 180,E1 -17433.598,E2 -17433.598} C_VEL
LIN {X 0,Y 283.286,Z 357.96,A -85,B 0,C 180,E1 -17437.768,E2 -17437.768} C_VEL
LIN {X 0,Y 286.757,Z 367.467,A -85,B 0,C 180,E1 -17439.557,E2 -17439.557} C_VEL
LIN {X 0,Y 288.783,Z 375.927,A -85,B 0,C 180,E1 -17441.229,E2 -17441.229} C_VEL
LIN {X 0,Y 289.539,Z 381.747,A -85,B 0,C 180,E1 -17442.426,E2 -17442.426} C_VEL
LIN {X 0,Y 287.931,Z 388.558,A -85,B 0,C 180,E1 -17443.696,E2 -17443.696} C_VEL
LIN {X 0,Y 286.043,Z 394.544,A -85,B 0,C 180,E1 -17445.048,E2 -17445.048} C_VEL
LIN {X 0,Y 284.405,Z 399.208,A -85,B 0,C 180,E1 -17446.421,E2 -17446.421} C_VEL
LIN {X 0,Y 282.988,Z 402.905,A -85,B 0,C 180,E1 -17447.812,E2 -17447.812} C_VEL
LIN {X 0,Y 281.627,Z 405.782,A -85,B 0,C 180,E1 -17449.211,E2 -17449.211} C_VEL
LIN {X 0,Y 279.81,Z 408.671,A -85,B 0,C 180,E1 -17451.331,E2 -17451.331} C_VEL
LIN {X 0,Y 278.665,Z 409.723,A -85,B 0,C 180,E1 -17452.754,E2 -17452.754} C_VEL
LIN {X 0,Y 277.744,Z 410.099,A -85,B 0,C 180,E1 -17454.189,E2 -17454.189} C_VEL
LIN {X 0,Y 277.021,Z 409.805,A -85,B 0,C 180,E1 -17455.633,E2 -17455.633} C_VEL
LIN {X 0,Y 276.518,Z 408.832,A -85,B 0,C 180,E1 -17457.084,E2 -17457.084} C_VEL
LIN {X 0,Y 276.092,Z 406.114,A -85,B 0,C 180,E1 -17459.269,E2 -17459.269} C_VEL
LIN {X 0,Y 275.854,Z 401.721,A -85,B 0,C 180,E1 -17461.458,E2 -17461.458} C_VEL
LIN {X 0,Y 275.954,Z 396.555,A -85,B 0,C 180,E1 -17463.283,E2 -17463.283} C_VEL
LIN {X 0,Y 276.285,Z 389.79,A -85,B 0,C 180,E1 -17465.106,E2 -17465.106} C_VEL
LIN {X 0,Y 276.522,Z 382.724,A -85,B 0,C 180,E1 -17466.565,E2 -17466.565} C_VEL
LIN {X 0,Y 276.746,Z 373.693,A -85,B 0,C 180,E1 -17468.026,E2 -17468.026} C_VEL
LIN {X 0,Y 276.962,Z 364.914,A -85,B 0,C 180,E1 -17469.123,E2 -17469.123} C_VEL
LIN {X 0,Y 277.194,Z 354.963,A -85,B 0,C 180,E1 -17470.036,E2 -17470.036} C_VEL
LIN {X 0,Y 276.62,Z 349.95,A -85,B 0,C 180,E1 -17470.427,E2 -17470.427} C_VEL
LIN {X 0,Y 276.685,Z 340.123,A -85,B 0,C 180,E1 -17475.153,E2 -17475.153} C_VEL
LIN {X 0,Y 276.821,Z 331.701,A -85,B 0,C 180,E1 -17479.269,E2 -17479.269} C_VEL
LIN {X 0,Y 277.011,Z 323.853,A -85,B 0,C 180,E1 -17483.154,E2 -17483.154} C_VEL
LIN {X 0,Y 277.294,Z 315.857,A -85,B 0,C 180,E1 -17487.14,E2 -17487.14} C_VEL
LIN {X 0,Y 277.498,Z 309.916,A -85,B 0,C 180,E1 -17490.22,E2 -17490.22} C_VEL
LIN {X 0,Y 277.272,Z 309.945,A -85,B 0,C 180,E1 -17495.658,E2 -17495.658} C_VEL
LIN {X 0,Y 277.21,Z 309.955,A -85,B 0,C 180,E1 -17499.329,E2 -17499.329} C_VEL
LIN {X 0,Y 277.193,Z 309.957,A -85,B 0,C 180,E1 -17503.198,E2 -17503.198} C_VEL
LIN {X 0,Y 277.207,Z 309.954,A -85,B 0,C 180,E1 -17507.323,E2 -17507.323} C_VEL
LIN {X 0,Y 277.257,Z 309.945,A -85,B 0,C 180,E1 -17511.791,E2 -17511.791} C_VEL
LIN {X 0,Y 277.276,Z 309.945,A -85,B 0,C 180,E1 -17514.34,E2 -17514.34} C_VEL
LIN {X 0,Y 277.236,Z 309.948,A -85,B 0,C 180,E1 -17517.835,E2 -17517.835} C_VEL
LIN {X 0,Y 277.28,Z 309.944,A -85,B 0,C 180,E1 -17521.211,E2 -17521.211} C_VEL
LIN {X 0,Y 277.304,Z 309.944,A -85,B 0,C 180,E1 -17524.478,E2 -17524.478} C_VEL
LIN {X 0,Y 277.281,Z 309.942,A -85,B 0,C 180,E1 -17527.654,E2 -17527.654} C_VEL
LIN {X 0,Y 277.335,Z 309.938,A -85,B 0,C 180,E1 -17530.765,E2 -17530.765} C_VEL
LIN {X 0,Y 277.424,Z 309.925,A -85,B 0,C 180,E1 -17535.325,E2 -17535.325} C_VEL
LIN {X 0,Y 277.446,Z 309.924,A -85,B 0,C 180,E1 -17539.786,E2 -17539.786} C_VEL
LIN {X 0,Y 277.589,Z 309.905,A -85,B 0,C 180,E1 -17542.727,E2 -17542.727} C_VEL
LIN {X 0,Y 277.792,Z 309.88,A -85,B 0,C 180,E1 -17548.55,E2 -17548.55} C_VEL
LIN {X 0,Y 277.793,Z 309.88,A -85,B 0,C 180,E1 -17551.45,E2 -17551.45} C_VEL
LIN {X 0,Y 277.589,Z 309.905,A -85,B 0,C 180,E1 -17557.273,E2 -17557.273} C_VEL
LIN {X 0,Y 277.446,Z 309.924,A -85,B 0,C 180,E1 -17560.214,E2 -17560.214} C_VEL
LIN {X 0,Y 277.424,Z 309.925,A -85,B 0,C 180,E1 -17564.675,E2 -17564.675} C_VEL
LIN {X 0,Y 277.335,Z 309.938,A -85,B 0,C 180,E1 -17569.235,E2 -17569.235} C_VEL
LIN {X 0,Y 277.319,Z 309.94,A -85,B 0,C 180,E1 -17573.922,E2 -17573.922} C_VEL
LIN {X 0,Y 277.316,Z 309.942,A -85,B 0,C 180,E1 -17577.506,E2 -17577.506} C_VEL
LIN {X 0,Y 277.263,Z 309.944,A -85,B 0,C 180,E1 -17580.483,E2 -17580.483} C_VEL
LIN {X 0,Y 277.238,Z 309.949,A -85,B 0,C 180,E1 -17583.897,E2 -17583.897} C_VEL
LIN {X 0,Y 277.26,Z 309.947,A -85,B 0,C 180,E1 -17587.471,E2 -17587.471} C_VEL
LIN {X 0,Y 277.202,Z 309.957,A -85,B 0,C 180,E1 -17591.238,E2 -17591.238} C_VEL
LIN {X 0,Y 277.193,Z 309.956,A -85,B 0,C 180,E1 -17595.228,E2 -17595.228} C_VEL
LIN {X 0,Y 277.19,Z 309.955,A -85,B 0,C 180,E1 -17599.52,E2 -17599.52} C_VEL
LIN {X 0,Y 277.249,Z 309.95,A -85,B 0,C 180,E1 -17602.531,E2 -17602.531} C_VEL
LIN {X 0,Y 277.332,Z 309.94,A -85,B 0,C 180,E1 -17606.748,E2 -17606.748} C_VEL
LIN {X 0,Y 277.529,Z 310.028,A -85,B 0,C 180,E1 -17608.184,E2 -17608.184} C_VEL
LIN {X 0,Y 277.57,Z 313.158,A -85,B 0,C 180,E1 -17610.416,E2 -17610.416} C_VEL
LIN {X 0,Y 277.067,Z 319.009,A -85,B 0,C 180,E1 -17614.458,E2 -17614.458} C_VEL
LIN {X 0,Y 276.67,Z 324.812,A -85,B 0,C 180,E1 -17618.39,E2 -17618.39} C_VEL
LIN {X 0,Y 276.306,Z 330.593,A -85,B 0,C 180,E1 -17622.23,E2 -17622.23} C_VEL
LIN {X 0,Y 276.077,Z 336.407,A -85,B 0,C 180,E1 -17626.022,E2 -17626.022} C_VEL
LIN {X 0,Y 276.033,Z 338.58,A -85,B 0,C 180,E1 -17627.363,E2 -17627.363} C_VEL
LIN {X 0,Y 277.121,Z 351.037,A -85,B 0,C 180,E1 -17628.389,E2 -17628.389} C_VEL
LIN {X 0,Y 277.782,Z 357.519,A -85,B 0,C 180,E1 -17629.064,E2 -17629.064} C_VEL
LIN {X 0,Y 277.297,Z 367.633,A -85,B 0,C 180,E1 -17630.336,E2 -17630.336} C_VEL
LIN {X 0,Y 276.827,Z 377.638,A -85,B 0,C 180,E1 -17631.942,E2 -17631.942} C_VEL
LIN {X 0,Y 276.55,Z 386.767,A -85,B 0,C 180,E1 -17633.802,E2 -17633.802} C_VEL
LIN {X 0,Y 276.149,Z 393.818,A -85,B 0,C 180,E1 -17635.623,E2 -17635.623} C_VEL
LIN {X 0,Y 275.904,Z 400.389,A -85,B 0,C 180,E1 -17637.812,E2 -17637.812} C_VEL
LIN {X 0,Y 275.993,Z 405.173,A -85,B 0,C 180,E1 -17640.002,E2 -17640.002} C_VEL
LIN {X 0,Y 276.211,Z 407.499,A -85,B 0,C 180,E1 -17641.46,E2 -17641.46} C_VEL
LIN {X 0,Y 276.548,Z 409.2,A -85,B 0,C 180,E1 -17642.915,E2 -17642.915} C_VEL
LIN {X 0,Y 277.04,Z 410.299,A -85,B 0,C 180,E1 -17644.367,E2 -17644.367} C_VEL
LIN {X 0,Y 277.738,Z 410.788,A -85,B 0,C 180,E1 -17645.811,E2 -17645.811} C_VEL
LIN {X 0,Y 278.639,Z 410.66,A -85,B 0,C 180,E1 -17647.247,E2 -17647.247} C_VEL
LIN {X 0,Y 279.781,Z 409.87,A -85,B 0,C 180,E1 -17648.753,E2 -17648.753} C_VEL
LIN {X 0,Y 281.032,Z 408.631,A -85,B 0,C 180,E1 -17650.084,E2 -17650.084} C_VEL
LIN {X 0,Y 283.172,Z 405.535,A -85,B 0,C 180,E1 -17652.18,E2 -17652.18} C_VEL
LIN {X 0,Y 285.615,Z 401.067,A -85,B 0,C 180,E1 -17654.247,E2 -17654.247} C_VEL
LIN {X 0,Y 285.976,Z 400.329,A -85,B 0,C 180,E1 -17654.519,E2 -17654.519} C_VEL
LIN {X 0,Y 287.031,Z 396.679,A -85,B 0,C 180,E1 -17655.9,E2 -17655.9} C_VEL
LIN {X 0,Y 287.027,Z 393.011,A -85,B 0,C 180,E1 -17657.3,E2 -17657.3} C_VEL
LIN {X 0,Y 286.603,Z 389.132,A -85,B 0,C 180,E1 -17658.694,E2 -17658.694} C_VEL
LIN {X 0,Y 286.392,Z 384.84,A -85,B 0,C 180,E1 -17660.041,E2 -17660.041} C_VEL
LIN {X 0,Y 286.156,Z 377.746,A -85,B 0,C 180,E1 -17662.071,E2 -17662.071} C_VEL
LIN {X 0,Y 285.023,Z 370.49,A -85,B 0,C 180,E1 -17664.17,E2 -17664.17} C_VEL
LIN {X 0,Y 283.035,Z 362.408,A -85,B 0,C 180,E1 -17666.631,E2 -17666.631} C_VEL
LIN {X 0,Y 279.987,Z 353.742,A -85,B 0,C 180,E1 -17669.675,E2 -17669.675} C_VEL
LIN {X 0,Y 278.501,Z 351.236,A -85,B 0,C 180,E1 -17670.907,E2 -17670.907} C_VEL
LIN {X 0,Y 277.841,Z 349.051,A -85,B 0,C 180,E1 -17671.768,E2 -17671.768} C_VEL
LIN {X 0,Y 278.317,Z 348.297,A -85,B 0,C 180,E1 -17673.75,E2 -17673.75} C_VEL
LIN {X 0,Y 278.691,Z 347.749,A -85,B 0,C 180,E1 -17676.198,E2 -17676.198} C_VEL
LIN {X 0,Y 279.01,Z 347.619,A -85,B 0,C 180,E1 -17679.032,E2 -17679.032} C_VEL
LIN {X 0,Y 279.438,Z 348.26,A -85,B 0,C 180,E1 -17682.772,E2 -17682.772} C_VEL
LIN {X 0,Y 280.033,Z 349.948,A -85,B 0,C 180,E1 -17686.706,E2 -17686.706} C_VEL
LIN {X 0,Y 280.496,Z 351.743,A -85,B 0,C 180,E1 -17689.349,E2 -17689.349} C_VEL
LIN {X 0,Y 281.203,Z 355.184,A -85,B 0,C 180,E1 -17693.11,E2 -17693.11} C_VEL
LIN {X 0,Y 281.6,Z 357.075,A -85,B 0,C 180,E1 -17694.687,E2 -17694.687} C_VEL
LIN {X 0,Y 283.562,Z 361.413,A -85,B 0,C 180,E1 -17695.974,E2 -17695.974} C_VEL
LIN {X 0,Y 284.403,Z 362.801,A -85,B 0,C 180,E1 -17696.436,E2 -17696.436} C_VEL
LIN {X 0,Y 286.026,Z 372.076,A -85,B 0,C 180,E1 -17698.187,E2 -17698.187} C_VEL
LIN {X 0,Y 287.206,Z 384.523,A -85,B 0,C 180,E1 -17700.345,E2 -17700.345} C_VEL
LIN {X 0,Y 287.165,Z 394.592,A -85,B 0,C 180,E1 -17702.041,E2 -17702.041} C_VEL
LIN {X 0,Y 286.246,Z 403.35,A -85,B 0,C 180,E1 -17703.522,E2 -17703.522} C_VEL
LIN {X 0,Y 284.568,Z 410.745,A -85,B 0,C 180,E1 -17704.784,E2 -17704.784} C_VEL
LIN {X 0,Y 280.862,Z 421.332,A -85,B 0,C 180,E1 -17706.789,E2 -17706.789} C_VEL
LIN {X 0,Y 277.544,Z 429.968,A -85,B 0,C 180,E1 -17708.848,E2 -17708.848} C_VEL
